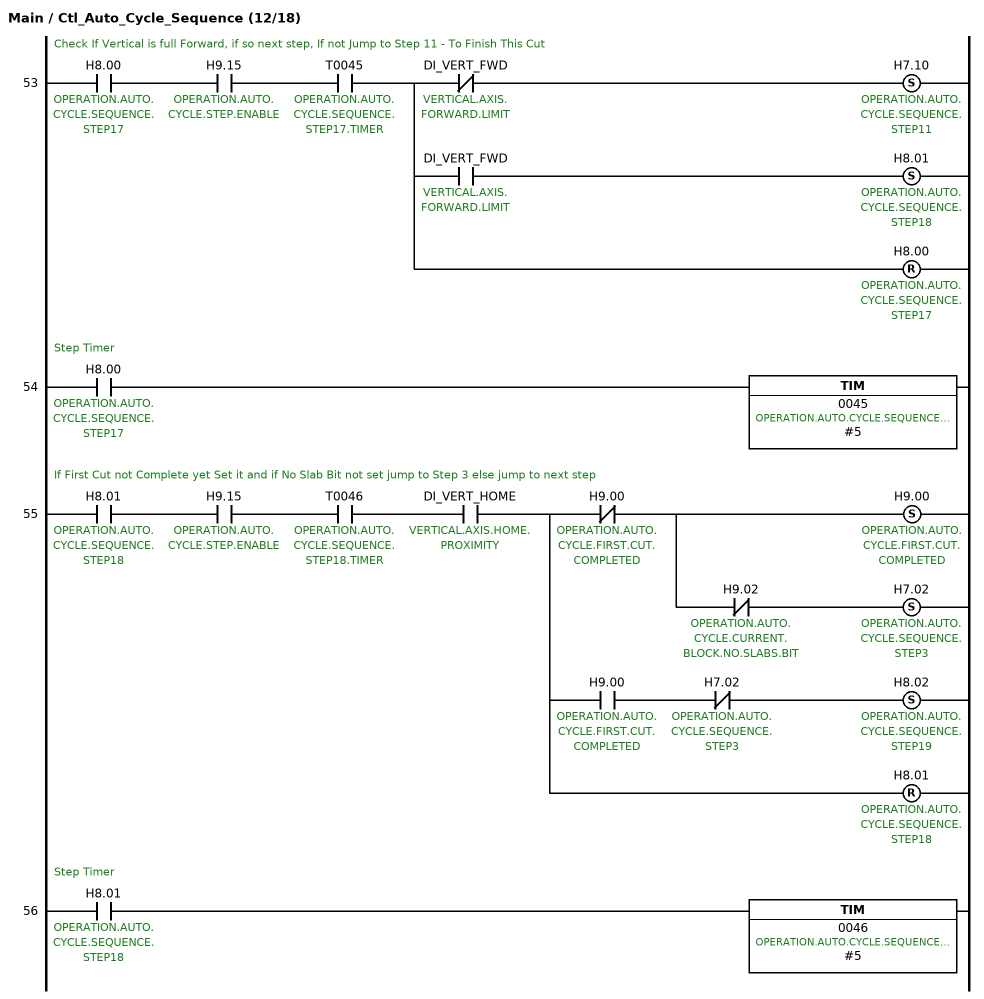
; [picture p24: Main / Ctl_Auto_Cycle_Sequence, rungs 53-56]
; rung 53: Check If Vertical is full Forward, if so next step, If not Jump to Step 11 - To Finish This Cut
LD H8.00  ; OPERATION.AUTO.CYCLE.SEQUENCE.STEP17
AND H9.15  ; OPERATION.AUTO.CYCLE.STEP.ENABLE
AND T0045  ; OPERATION.AUTO.CYCLE.SEQUENCE.STEP17.TIMER
OUT TR0
ANDNOT DI_VERT_FWD  ; VERTICAL.AXIS.FORWARD.LIMIT
SET H7.10  ; OPERATION.AUTO.CYCLE.SEQUENCE.STEP11
LD TR0
AND DI_VERT_FWD  ; VERTICAL.AXIS.FORWARD.LIMIT
SET H8.01  ; OPERATION.AUTO.CYCLE.SEQUENCE.STEP18
LD TR0
RSET H8.00  ; OPERATION.AUTO.CYCLE.SEQUENCE.STEP17
; rung 54: Step Timer
LD H8.00  ; OPERATION.AUTO.CYCLE.SEQUENCE.STEP17
TIM 0045 #5  ; OPERATION.AUTO.CYCLE.SEQUENCE.STEP17.TIMER
; rung 55: If First Cut not Complete yet Set it and if No Slab Bit not set jump to Step 3 else jump to next step
LD H8.01  ; OPERATION.AUTO.CYCLE.SEQUENCE.STEP18
AND H9.15  ; OPERATION.AUTO.CYCLE.STEP.ENABLE
AND T0046  ; OPERATION.AUTO.CYCLE.SEQUENCE.STEP18.TIMER
AND DI_VERT_HOME  ; VERTICAL.AXIS.HOME.PROXIMITY
OUT TR0
ANDNOT H9.00  ; OPERATION.AUTO.CYCLE.FIRST.CUT.COMPLETED
SET H9.00  ; OPERATION.AUTO.CYCLE.FIRST.CUT.COMPLETED
ANDNOT H9.02  ; OPERATION.AUTO.CYCLE.CURRENT.BLOCK.NO.SLABS.BIT
SET H7.02  ; OPERATION.AUTO.CYCLE.SEQUENCE.STEP3
LD TR0
AND H9.00  ; OPERATION.AUTO.CYCLE.FIRST.CUT.COMPLETED
ANDNOT H7.02  ; OPERATION.AUTO.CYCLE.SEQUENCE.STEP3
SET H8.02  ; OPERATION.AUTO.CYCLE.SEQUENCE.STEP19
LD TR0
RSET H8.01  ; OPERATION.AUTO.CYCLE.SEQUENCE.STEP18
; rung 56: Step Timer
LD H8.01  ; OPERATION.AUTO.CYCLE.SEQUENCE.STEP18
TIM 0046 #5  ; OPERATION.AUTO.CYCLE.SEQUENCE.STEP18.TIMER

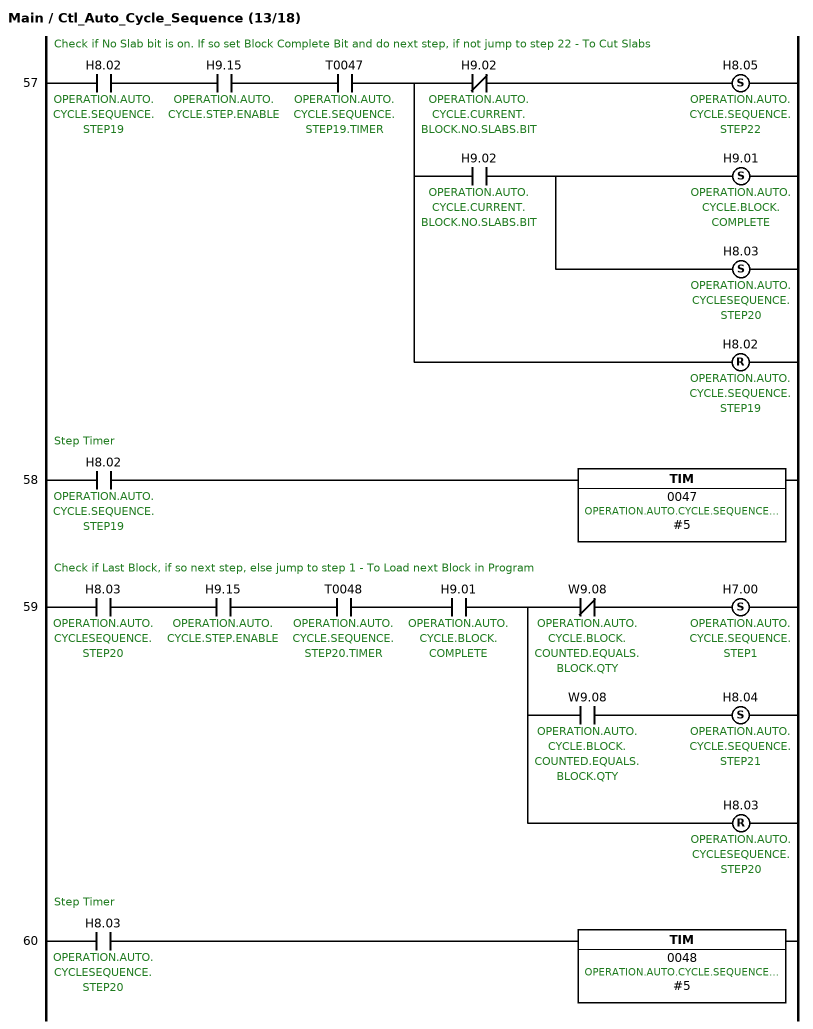
; rung 57: Check if No Slab bit is on. If so set Block Complete Bit and do next step, if not jump to step 22 - To Cut Slabs
LD H8.02  ; OPERATION.AUTO.CYCLE.SEQUENCE.STEP19
AND H9.15  ; OPERATION.AUTO.CYCLE.STEP.ENABLE
AND T0047  ; OPERATION.AUTO.CYCLE.SEQUENCE.STEP19.TIMER
OUT TR0
ANDNOT H9.02  ; OPERATION.AUTO.CYCLE.CURRENT.BLOCK.NO.SLABS.BIT
SET H8.05  ; OPERATION.AUTO.CYCLE.SEQUENCE.STEP22
LD TR0
AND H9.02  ; OPERATION.AUTO.CYCLE.CURRENT.BLOCK.NO.SLABS.BIT
SET H9.01  ; OPERATION.AUTO.CYCLE.BLOCK.COMPLETE
SET H8.03  ; OPERATION.AUTO.CYCLESEQUENCE.STEP20
LD TR0
RSET H8.02  ; OPERATION.AUTO.CYCLE.SEQUENCE.STEP19
; rung 58: Step Timer
LD H8.02  ; OPERATION.AUTO.CYCLE.SEQUENCE.STEP19
TIM 0047 #5  ; OPERATION.AUTO.CYCLE.SEQUENCE.STEP19.TIMER
; rung 59: Check if Last Block, if so next step, else jump to step 1 - To Load next Block in Program
LD H8.03  ; OPERATION.AUTO.CYCLESEQUENCE.STEP20
AND H9.15  ; OPERATION.AUTO.CYCLE.STEP.ENABLE
AND T0048  ; OPERATION.AUTO.CYCLE.SEQUENCE.STEP20.TIMER
AND H9.01  ; OPERATION.AUTO.CYCLE.BLOCK.COMPLETE
OUT TR0
ANDNOT W9.08  ; OPERATION.AUTO.CYCLE.BLOCK.COUNTED.EQUALS.BLOCK.QTY
SET H7.00  ; OPERATION.AUTO.CYCLE.SEQUENCE.STEP1
LD TR0
AND W9.08  ; OPERATION.AUTO.CYCLE.BLOCK.COUNTED.EQUALS.BLOCK.QTY
SET H8.04  ; OPERATION.AUTO.CYCLE.SEQUENCE.STEP21
LD TR0
RSET H8.03  ; OPERATION.AUTO.CYCLESEQUENCE.STEP20
; rung 60: Step Timer
LD H8.03  ; OPERATION.AUTO.CYCLESEQUENCE.STEP20
TIM 0048 #5  ; OPERATION.AUTO.CYCLE.SEQUENCE.STEP20.TIMER

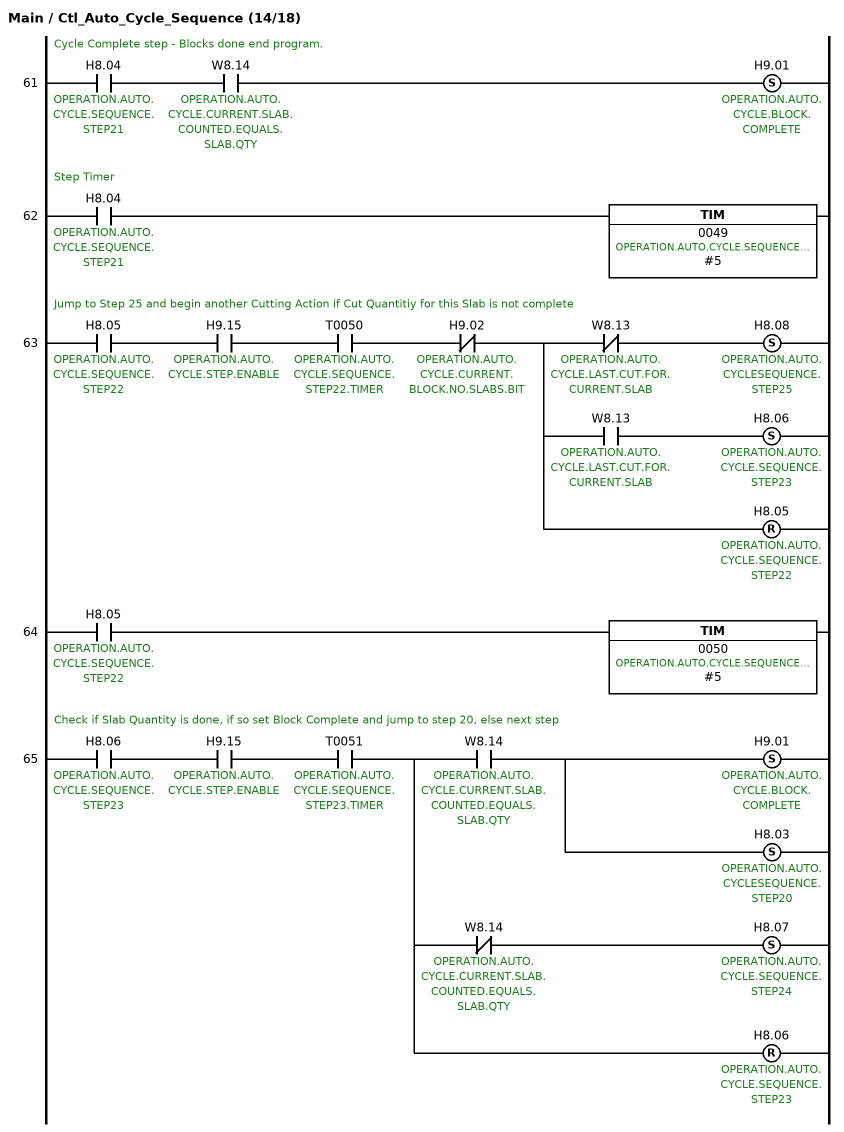
; rung 61: Cycle Complete step - Blocks done end program.
LD H8.04  ; OPERATION.AUTO.CYCLE.SEQUENCE.STEP21
AND W8.14  ; OPERATION.AUTO.CYCLE.CURRENT.SLAB.COUNTED.EQUALS.SLAB.QTY
SET H9.01  ; OPERATION.AUTO.CYCLE.BLOCK.COMPLETE
; rung 62: Step Timer
LD H8.04  ; OPERATION.AUTO.CYCLE.SEQUENCE.STEP21
TIM 0049 #5  ; OPERATION.AUTO.CYCLE.SEQUENCE.STEP21.TIMER
; rung 63: Jump to Step 25 and begin another Cutting Action if Cut Quantitiy for this Slab is not complete
LD H8.05  ; OPERATION.AUTO.CYCLE.SEQUENCE.STEP22
AND H9.15  ; OPERATION.AUTO.CYCLE.STEP.ENABLE
AND T0050  ; OPERATION.AUTO.CYCLE.SEQUENCE.STEP22.TIMER
ANDNOT H9.02  ; OPERATION.AUTO.CYCLE.CURRENT.BLOCK.NO.SLABS.BIT
OUT TR0
ANDNOT W8.13  ; OPERATION.AUTO.CYCLE.LAST.CUT.FOR.CURRENT.SLAB
SET H8.08  ; OPERATION.AUTO.CYCLESEQUENCE.STEP25
LD TR0
AND W8.13  ; OPERATION.AUTO.CYCLE.LAST.CUT.FOR.CURRENT.SLAB
SET H8.06  ; OPERATION.AUTO.CYCLE.SEQUENCE.STEP23
LD TR0
RSET H8.05  ; OPERATION.AUTO.CYCLE.SEQUENCE.STEP22
; rung 64
LD H8.05  ; OPERATION.AUTO.CYCLE.SEQUENCE.STEP22
TIM 0050 #5  ; OPERATION.AUTO.CYCLE.SEQUENCE.STEP22.TIMER
; rung 65: Check if Slab Quantity is done, if so set Block Complete and jump to step 20, else next step
LD H8.06  ; OPERATION.AUTO.CYCLE.SEQUENCE.STEP23
AND H9.15  ; OPERATION.AUTO.CYCLE.STEP.ENABLE
AND T0051  ; OPERATION.AUTO.CYCLE.SEQUENCE.STEP23.TIMER
OUT TR0
AND W8.14  ; OPERATION.AUTO.CYCLE.CURRENT.SLAB.COUNTED.EQUALS.SLAB.QTY
SET H9.01  ; OPERATION.AUTO.CYCLE.BLOCK.COMPLETE
SET H8.03  ; OPERATION.AUTO.CYCLESEQUENCE.STEP20
LD TR0
ANDNOT W8.14  ; OPERATION.AUTO.CYCLE.CURRENT.SLAB.COUNTED.EQUALS.SLAB.QTY
SET H8.07  ; OPERATION.AUTO.CYCLE.SEQUENCE.STEP24
LD TR0
RSET H8.06  ; OPERATION.AUTO.CYCLE.SEQUENCE.STEP23

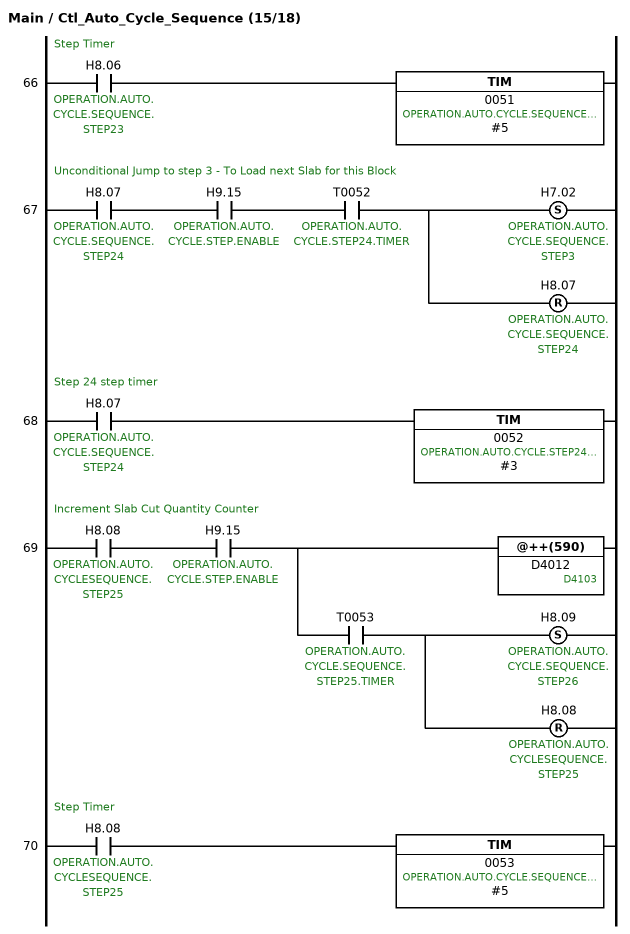
; rung 66: Step Timer
LD H8.06  ; OPERATION.AUTO.CYCLE.SEQUENCE.STEP23
TIM 0051 #5  ; OPERATION.AUTO.CYCLE.SEQUENCE.STEP23.TIMER
; rung 67: Unconditional Jump to step 3 - To Load next Slab for this Block
LD H8.07  ; OPERATION.AUTO.CYCLE.SEQUENCE.STEP24
AND H9.15  ; OPERATION.AUTO.CYCLE.STEP.ENABLE
AND T0052  ; OPERATION.AUTO.CYCLE.STEP24.TIMER
SET H7.02  ; OPERATION.AUTO.CYCLE.SEQUENCE.STEP3
RSET H8.07  ; OPERATION.AUTO.CYCLE.SEQUENCE.STEP24
; rung 68: Step 24 step timer
LD H8.07  ; OPERATION.AUTO.CYCLE.SEQUENCE.STEP24
TIM 0052 #3  ; OPERATION.AUTO.CYCLE.STEP24.TIMER
; rung 69: Increment Slab Cut Quantity Counter
LD H8.08  ; OPERATION.AUTO.CYCLESEQUENCE.STEP25
AND H9.15  ; OPERATION.AUTO.CYCLE.STEP.ENABLE
@++(590) D4012  ; D4103
AND T0053  ; OPERATION.AUTO.CYCLE.SEQUENCE.STEP25.TIMER
SET H8.09  ; OPERATION.AUTO.CYCLE.SEQUENCE.STEP26
RSET H8.08  ; OPERATION.AUTO.CYCLESEQUENCE.STEP25
; rung 70: Step Timer
LD H8.08  ; OPERATION.AUTO.CYCLESEQUENCE.STEP25
TIM 0053 #5  ; OPERATION.AUTO.CYCLE.SEQUENCE.STEP25.TIMER

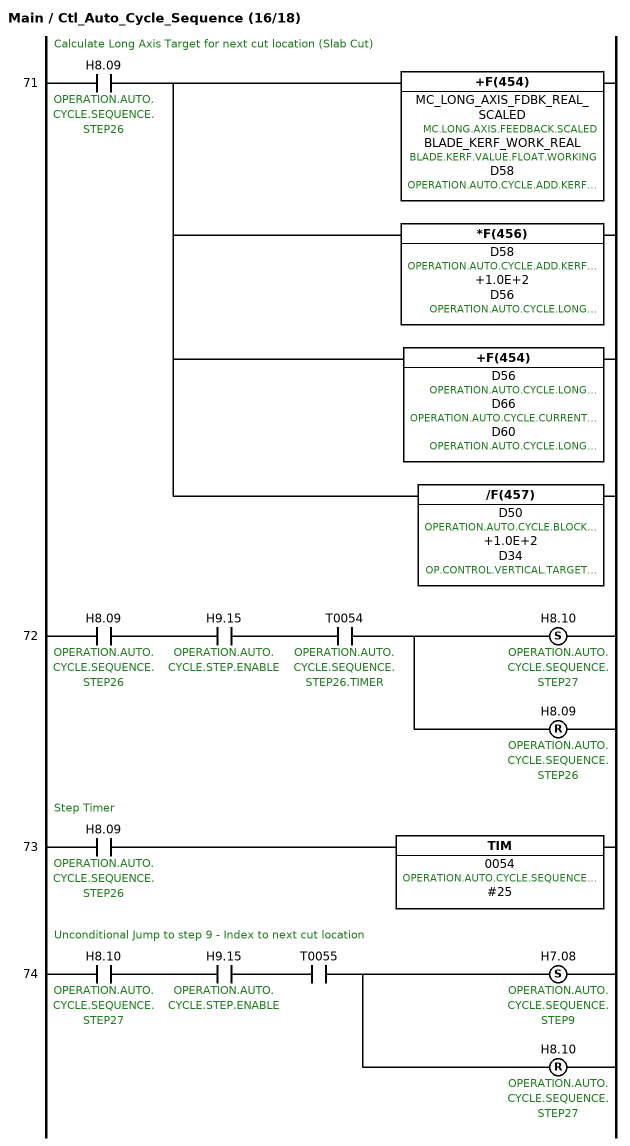
; rung 71: Calculate Long Axis Target for next cut location (Slab Cut)
LD H8.09  ; OPERATION.AUTO.CYCLE.SEQUENCE.STEP26
+F(454) MC_LONG_AXIS_FDBK_REAL_SCALED BLADE_KERF_WORK_REAL D58  ; MC.LONG.AXIS.FEEDBACK.SCALED, BLADE.KERF.VALUE.FLOAT.WORKING, OPERATION.AUTO.CYCLE.ADD.KERF.TO.LOCATION.REAL
*F(456) D58 +1.0E+2 D56  ; OPERATION.AUTO.CYCLE.ADD.KERF.TO.LOCATION.REAL, OPERATION.AUTO.CYCLE.LONG.TARGET.KERF
+F(454) D56 D66 D60  ; OPERATION.AUTO.CYCLE.LONG.TARGET.KERF, OPERATION.AUTO.CYCLE.CURRENT.SLAB.SIZE.REAL.RAW, OPERATION.AUTO.CYCLE.LONG.INDEX.LOCATION.REAL
/F(457) D50 +1.0E+2 D34  ; OPERATION.AUTO.CYCLE.BLOCK.HEIGHT.REAL, OP.CONTROL.VERTICAL.TARGET.SCALED
; rung 72
LD H8.09  ; OPERATION.AUTO.CYCLE.SEQUENCE.STEP26
AND H9.15  ; OPERATION.AUTO.CYCLE.STEP.ENABLE
AND T0054  ; OPERATION.AUTO.CYCLE.SEQUENCE.STEP26.TIMER
SET H8.10  ; OPERATION.AUTO.CYCLE.SEQUENCE.STEP27
RSET H8.09  ; OPERATION.AUTO.CYCLE.SEQUENCE.STEP26
; rung 73: Step Timer
LD H8.09  ; OPERATION.AUTO.CYCLE.SEQUENCE.STEP26
TIM 0054 #25  ; OPERATION.AUTO.CYCLE.SEQUENCE.STEP26.TIMER
; rung 74: Unconditional Jump to step 9 - Index to next cut location
LD H8.10  ; OPERATION.AUTO.CYCLE.SEQUENCE.STEP27
AND H9.15  ; OPERATION.AUTO.CYCLE.STEP.ENABLE
AND T0055
SET H7.08  ; OPERATION.AUTO.CYCLE.SEQUENCE.STEP9
RSET H8.10  ; OPERATION.AUTO.CYCLE.SEQUENCE.STEP27

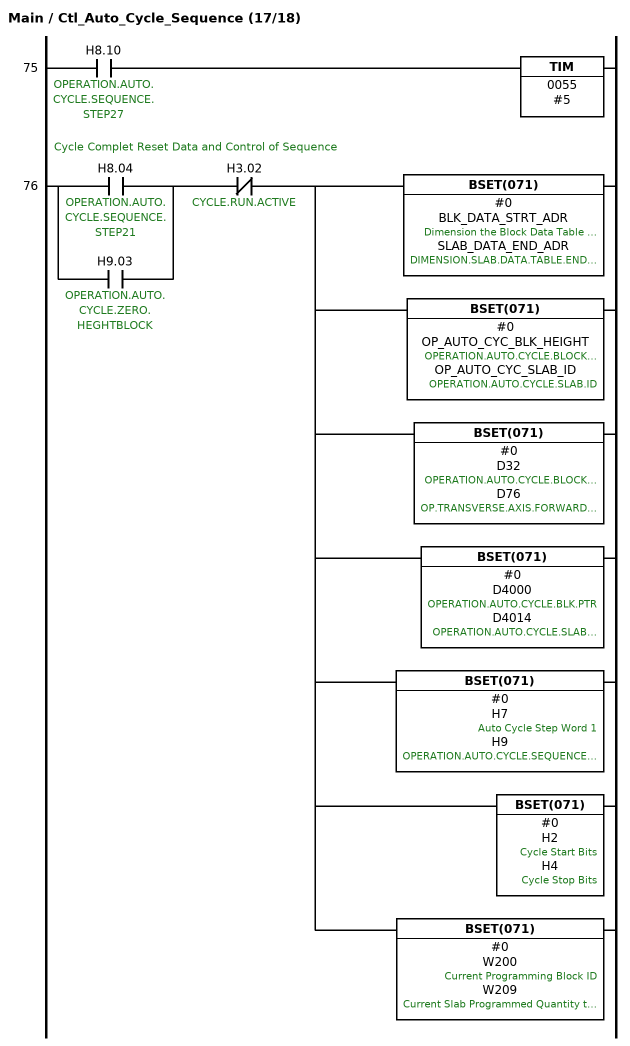
; rung 75
LD H8.10  ; OPERATION.AUTO.CYCLE.SEQUENCE.STEP27
TIM 0055 #5
; rung 76: Cycle Complet Reset Data and Control of Sequence
LD H8.04  ; OPERATION.AUTO.CYCLE.SEQUENCE.STEP21
OR H9.03  ; OPERATION.AUTO.CYCLE.ZERO.HEGHTBLOCK
ANDNOT H3.02  ; CYCLE.RUN.ACTIVE
BSET(071) #0 BLK_DATA_STRT_ADR SLAB_DATA_END_ADR  ; Dimension the Block Data Table - Start Address, DIMENSION.SLAB.DATA.TABLE.END.ADDRESS
BSET(071) #0 OP_AUTO_CYC_BLK_HEIGHT OP_AUTO_CYC_SLAB_ID  ; OPERATION.AUTO.CYCLE.BLOCK.HEIGHT.WORKING, OPERATION.AUTO.CYCLE.SLAB.ID
BSET(071) #0 D32 D76  ; OPERATION.AUTO.CYCLE.BLOCK.FIRST.CUT.WORKING.REAL, OP.TRANSVERSE.AXIS.FORWARD.TARGET
BSET(071) #0 D4000 D4014  ; OPERATION.AUTO.CYCLE.BLK.PTR, OPERATION.AUTO.CYCLE.SLAB.POINTER
BSET(071) #0 H7 H9  ; Auto Cycle Step Word 1, OPERATION.AUTO.CYCLE.SEQUENCE.STATE.BITS
BSET(071) #0 H2 H4  ; Cycle Start Bits, Cycle Stop Bits
BSET(071) #0 W200 W209  ; Current Programming Block ID, Current Slab Programmed Quantity to cut

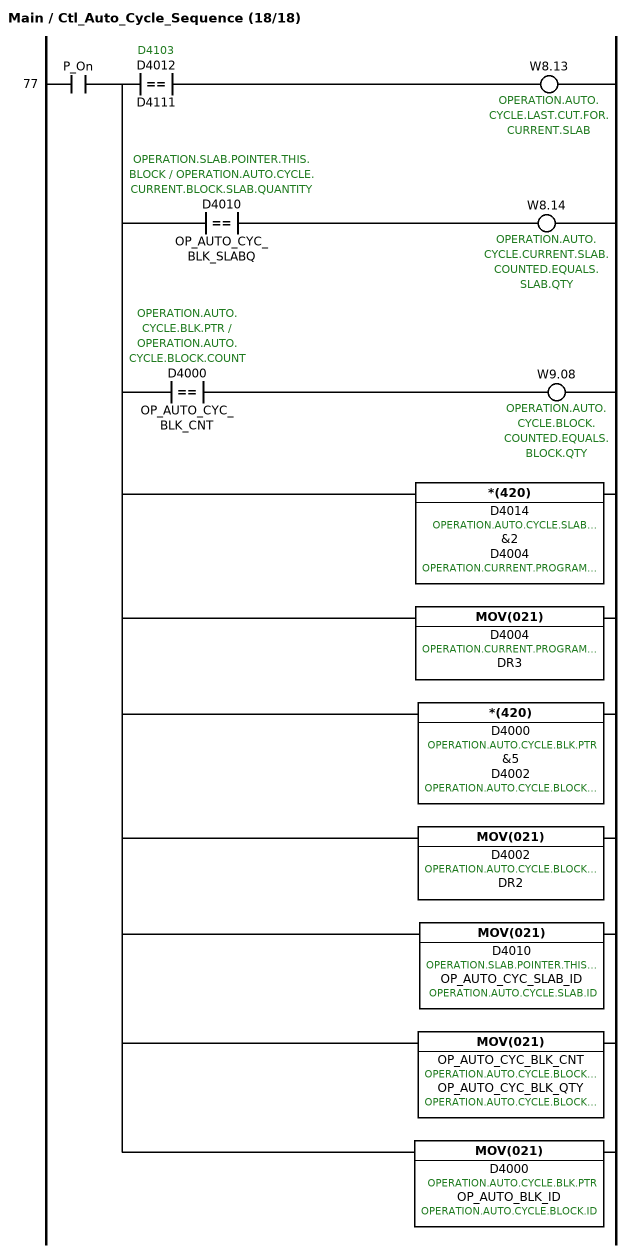
; rung 77
LD P_On
OUT TR0
AND=(300) D4012 D4111  ; D4103
OUT W8.13  ; OPERATION.AUTO.CYCLE.LAST.CUT.FOR.CURRENT.SLAB
LD TR0
AND=(300) D4010 OP_AUTO_CYC_BLK_SLABQ  ; OPERATION.SLAB.POINTER.THIS.BLOCK, OPERATION.AUTO.CYCLE.CURRENT.BLOCK.SLAB.QUANTITY
OUT W8.14  ; OPERATION.AUTO.CYCLE.CURRENT.SLAB.COUNTED.EQUALS.SLAB.QTY
LD TR0
AND=(300) D4000 OP_AUTO_CYC_BLK_CNT  ; OPERATION.AUTO.CYCLE.BLK.PTR, OPERATION.AUTO.CYCLE.BLOCK.COUNT
OUT W9.08  ; OPERATION.AUTO.CYCLE.BLOCK.COUNTED.EQUALS.BLOCK.QTY
LD TR0
*(420) D4014 &2 D4004  ; OPERATION.AUTO.CYCLE.SLAB.POINTER, OPERATION.CURRENT.PROGRAM.SLAB.DATA.POINTER
MOV(021) D4004 DR3  ; OPERATION.CURRENT.PROGRAM.SLAB.DATA.POINTER
*(420) D4000 &5 D4002  ; OPERATION.AUTO.CYCLE.BLK.PTR, OPERATION.AUTO.CYCLE.BLOCK.DATA.POINTER
MOV(021) D4002 DR2  ; OPERATION.AUTO.CYCLE.BLOCK.DATA.POINTER
MOV(021) D4010 OP_AUTO_CYC_SLAB_ID  ; OPERATION.SLAB.POINTER.THIS.BLOCK, OPERATION.AUTO.CYCLE.SLAB.ID
MOV(021) OP_AUTO_CYC_BLK_CNT OP_AUTO_CYC_BLK_QTY  ; OPERATION.AUTO.CYCLE.BLOCK.COUNT, OPERATION.AUTO.CYCLE.BLOCK.QUANTITY
MOV(021) D4000 OP_AUTO_BLK_ID  ; OPERATION.AUTO.CYCLE.BLK.PTR, OPERATION.AUTO.CYCLE.BLOCK.ID

### Section Ctl_Master_Home

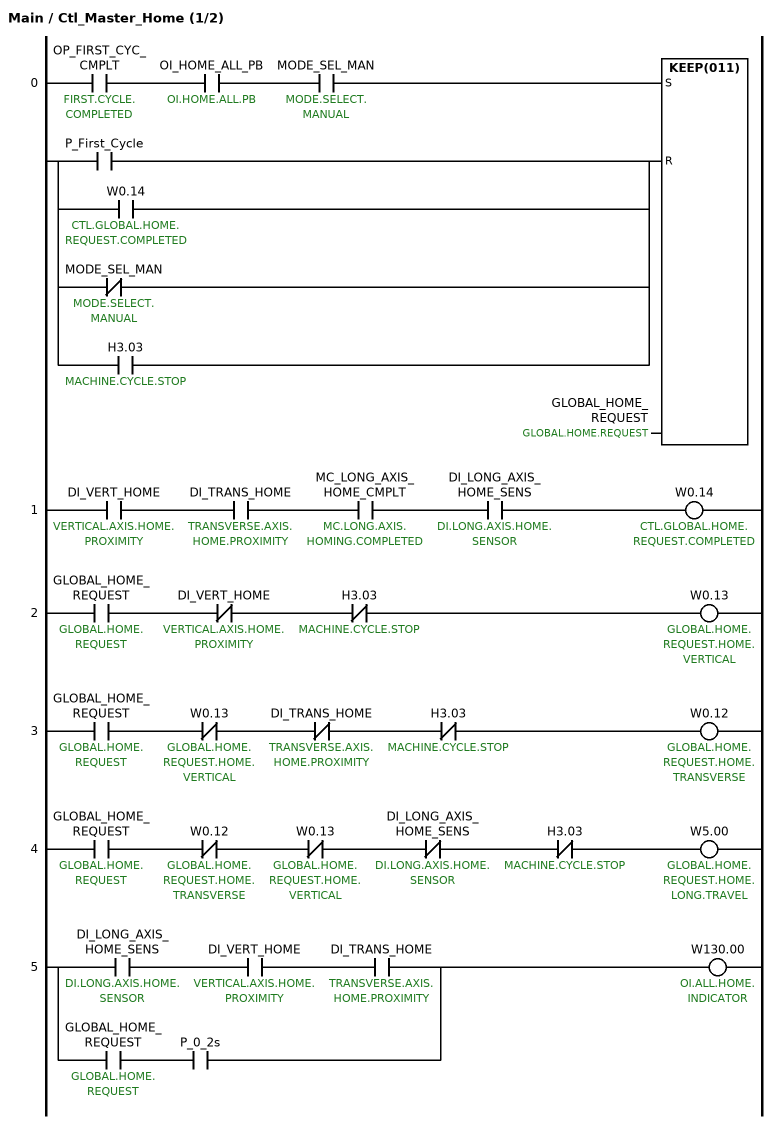
; rung 0
LD OP_FIRST_CYC_CMPLT  ; FIRST.CYCLE.COMPLETED
AND OI_HOME_ALL_PB  ; OI.HOME.ALL.PB
AND MODE_SEL_MAN  ; MODE.SELECT.MANUAL
LD P_First_Cycle
OR W0.14  ; CTL.GLOBAL.HOME.REQUEST.COMPLETED
ORNOT MODE_SEL_MAN  ; MODE.SELECT.MANUAL
OR H3.03  ; MACHINE.CYCLE.STOP
KEEP(011) GLOBAL_HOME_REQUEST  ; GLOBAL.HOME.REQUEST
; rung 1
LD DI_VERT_HOME  ; VERTICAL.AXIS.HOME.PROXIMITY
AND DI_TRANS_HOME  ; TRANSVERSE.AXIS.HOME.PROXIMITY
AND MC_LONG_AXIS_HOME_CMPLT  ; MC.LONG.AXIS.HOMING.COMPLETED
AND DI_LONG_AXIS_HOME_SENS  ; DI.LONG.AXIS.HOME.SENSOR
OUT W0.14  ; CTL.GLOBAL.HOME.REQUEST.COMPLETED
; rung 2
LD GLOBAL_HOME_REQUEST  ; GLOBAL.HOME.REQUEST
ANDNOT DI_VERT_HOME  ; VERTICAL.AXIS.HOME.PROXIMITY
ANDNOT H3.03  ; MACHINE.CYCLE.STOP
OUT W0.13  ; GLOBAL.HOME.REQUEST.HOME.VERTICAL
; rung 3
LD GLOBAL_HOME_REQUEST  ; GLOBAL.HOME.REQUEST
ANDNOT W0.13  ; GLOBAL.HOME.REQUEST.HOME.VERTICAL
ANDNOT DI_TRANS_HOME  ; TRANSVERSE.AXIS.HOME.PROXIMITY
ANDNOT H3.03  ; MACHINE.CYCLE.STOP
OUT W0.12  ; GLOBAL.HOME.REQUEST.HOME.TRANSVERSE
; rung 4
LD GLOBAL_HOME_REQUEST  ; GLOBAL.HOME.REQUEST
ANDNOT W0.12  ; GLOBAL.HOME.REQUEST.HOME.TRANSVERSE
ANDNOT W0.13  ; GLOBAL.HOME.REQUEST.HOME.VERTICAL
ANDNOT DI_LONG_AXIS_HOME_SENS  ; DI.LONG.AXIS.HOME.SENSOR
ANDNOT H3.03  ; MACHINE.CYCLE.STOP
OUT W5.00  ; GLOBAL.HOME.REQUEST.HOME.LONG.TRAVEL
; rung 5
LD DI_LONG_AXIS_HOME_SENS  ; DI.LONG.AXIS.HOME.SENSOR
AND DI_VERT_HOME  ; VERTICAL.AXIS.HOME.PROXIMITY
AND DI_TRANS_HOME  ; TRANSVERSE.AXIS.HOME.PROXIMITY
LD GLOBAL_HOME_REQUEST  ; GLOBAL.HOME.REQUEST
AND P_0_2s
ORLD
OUT W130.00  ; OI.ALL.HOME.INDICATOR

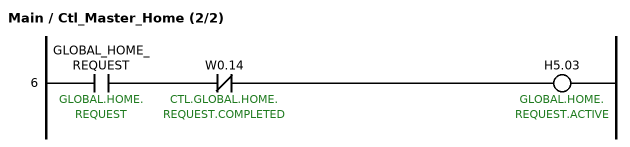
; rung 6
LD GLOBAL_HOME_REQUEST  ; GLOBAL.HOME.REQUEST
ANDNOT W0.14  ; CTL.GLOBAL.HOME.REQUEST.COMPLETED
OUT H5.03  ; GLOBAL.HOME.REQUEST.ACTIVE

### Section Ctl_Long_Axis

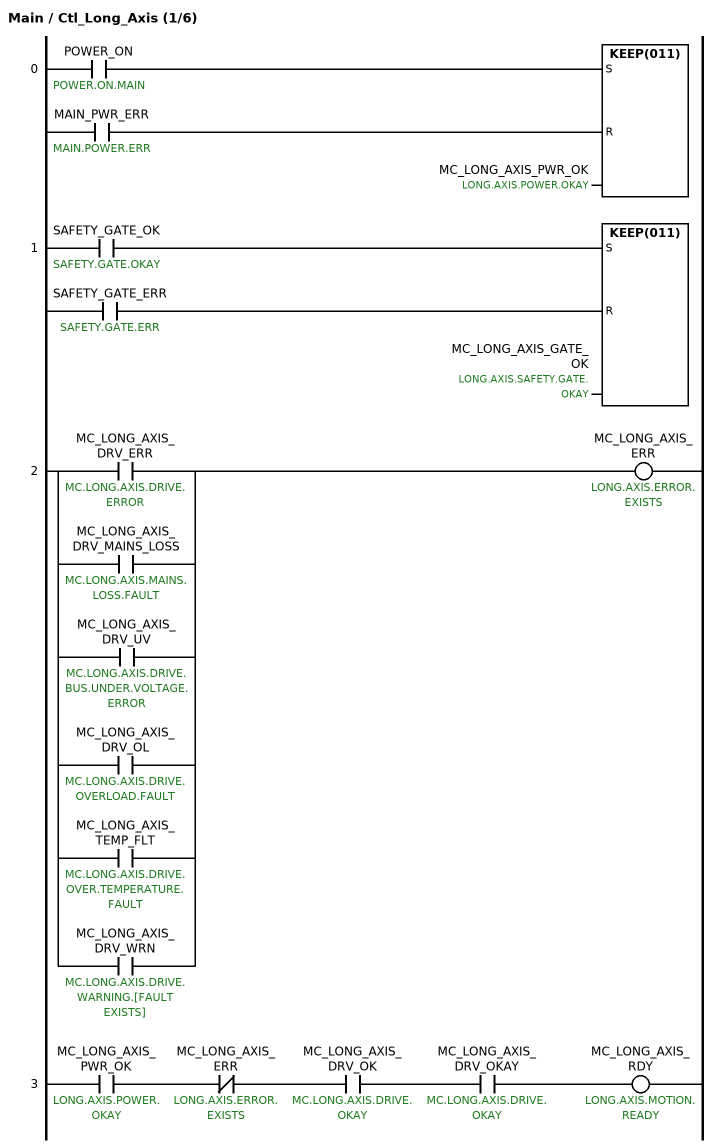
; rung 0
LD POWER_ON  ; POWER.ON.MAIN
LD MAIN_PWR_ERR  ; MAIN.POWER.ERR
KEEP(011) MC_LONG_AXIS_PWR_OK  ; LONG.AXIS.POWER.OKAY
; rung 1
LD SAFETY_GATE_OK  ; SAFETY.GATE.OKAY
LD SAFETY_GATE_ERR  ; SAFETY.GATE.ERR
KEEP(011) MC_LONG_AXIS_GATE_OK  ; LONG.AXIS.SAFETY.GATE.OKAY
; rung 2
LD MC_LONG_AXIS_DRV_ERR  ; MC.LONG.AXIS.DRIVE.ERROR
OR MC_LONG_AXIS_DRV_MAINS_LOSS  ; MC.LONG.AXIS.MAINS.LOSS.FAULT
OR MC_LONG_AXIS_DRV_UV  ; MC.LONG.AXIS.DRIVE.BUS.UNDER.VOLTAGE.ERROR
OR MC_LONG_AXIS_DRV_OL  ; MC.LONG.AXIS.DRIVE.OVERLOAD.FAULT
OR MC_LONG_AXIS_TEMP_FLT  ; MC.LONG.AXIS.DRIVE.OVER.TEMPERATURE.FAULT
OR MC_LONG_AXIS_DRV_WRN  ; MC.LONG.AXIS.DRIVE.WARNING.[FAULT EXISTS]
OUT MC_LONG_AXIS_ERR  ; LONG.AXIS.ERROR.EXISTS
; rung 3
LD MC_LONG_AXIS_PWR_OK  ; LONG.AXIS.POWER.OKAY
ANDNOT MC_LONG_AXIS_ERR  ; LONG.AXIS.ERROR.EXISTS
AND MC_LONG_AXIS_DRV_OK  ; MC.LONG.AXIS.DRIVE.OKAY
AND MC_LONG_AXIS_DRV_OKAY  ; MC.LONG.AXIS.DRIVE.OKAY
OUT MC_LONG_AXIS_RDY  ; LONG.AXIS.MOTION.READY

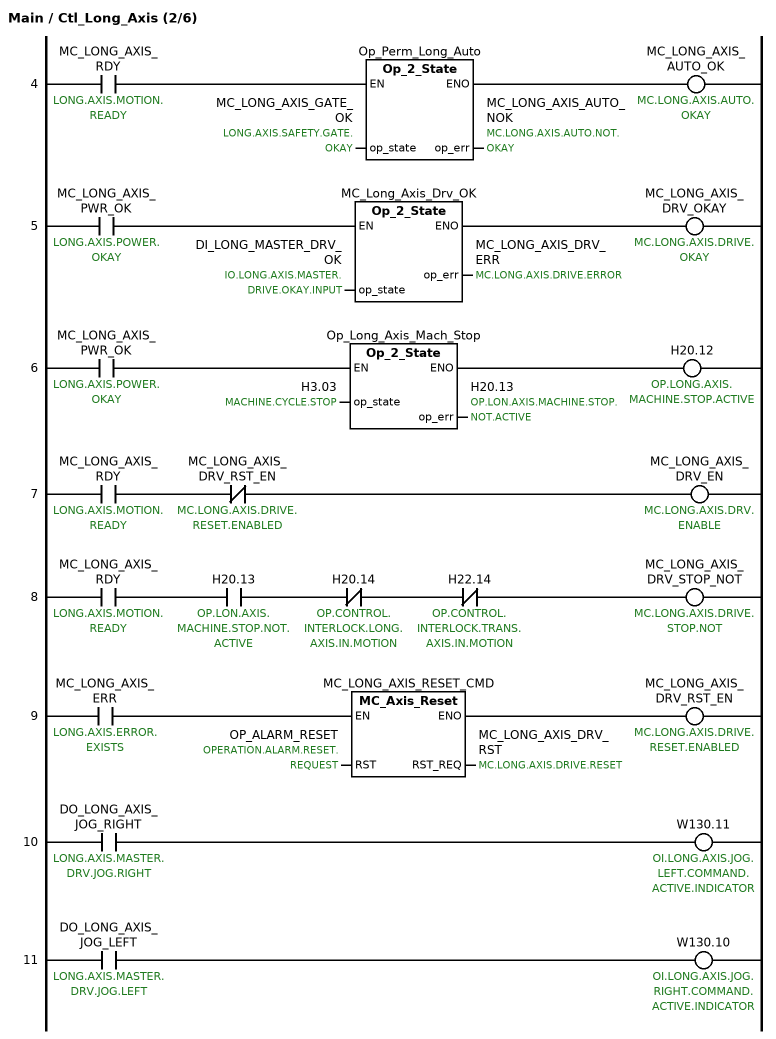
; rung 4
LD MC_LONG_AXIS_RDY  ; LONG.AXIS.MOTION.READY
CALL Op_Perm_Long_Auto : Op_2_State (op_state := MC_LONG_AXIS_GATE_OK, op_err => MC_LONG_AXIS_AUTO_NOK)  ; LONG.AXIS.SAFETY.GATE.OKAY, MC.LONG.AXIS.AUTO.NOT.OKAY
OUT MC_LONG_AXIS_AUTO_OK  ; MC.LONG.AXIS.AUTO.OKAY
; rung 5
LD MC_LONG_AXIS_PWR_OK  ; LONG.AXIS.POWER.OKAY
CALL MC_Long_Axis_Drv_OK : Op_2_State (op_state := DI_LONG_MASTER_DRV_OK, op_err => MC_LONG_AXIS_DRV_ERR)  ; IO.LONG.AXIS.MASTER.DRIVE.OKAY.INPUT, MC.LONG.AXIS.DRIVE.ERROR
OUT MC_LONG_AXIS_DRV_OKAY  ; MC.LONG.AXIS.DRIVE.OKAY
; rung 6
LD MC_LONG_AXIS_PWR_OK  ; LONG.AXIS.POWER.OKAY
CALL Op_Long_Axis_Mach_Stop : Op_2_State (op_state := H3.03, op_err => H20.13)  ; MACHINE.CYCLE.STOP, OP.LON.AXIS.MACHINE.STOP.NOT.ACTIVE
OUT H20.12  ; OP.LONG.AXIS.MACHINE.STOP.ACTIVE
; rung 7
LD MC_LONG_AXIS_RDY  ; LONG.AXIS.MOTION.READY
ANDNOT MC_LONG_AXIS_DRV_RST_EN  ; MC.LONG.AXIS.DRIVE.RESET.ENABLED
OUT MC_LONG_AXIS_DRV_EN  ; MC.LONG.AXIS.DRV.ENABLE
; rung 8
LD MC_LONG_AXIS_RDY  ; LONG.AXIS.MOTION.READY
AND H20.13  ; OP.LON.AXIS.MACHINE.STOP.NOT.ACTIVE
ANDNOT H20.14  ; OP.CONTROL.INTERLOCK.LONG.AXIS.IN.MOTION
ANDNOT H22.14  ; OP.CONTROL.INTERLOCK.TRANS.AXIS.IN.MOTION
OUT MC_LONG_AXIS_DRV_STOP_NOT  ; MC.LONG.AXIS.DRIVE.STOP.NOT
; rung 9
LD MC_LONG_AXIS_ERR  ; LONG.AXIS.ERROR.EXISTS
CALL MC_LONG_AXIS_RESET_CMD : MC_Axis_Reset (RST := OP_ALARM_RESET, RST_REQ => MC_LONG_AXIS_DRV_RST)  ; OPERATION.ALARM.RESET.REQUEST, MC.LONG.AXIS.DRIVE.RESET
OUT MC_LONG_AXIS_DRV_RST_EN  ; MC.LONG.AXIS.DRIVE.RESET.ENABLED
; rung 10
LD DO_LONG_AXIS_JOG_RIGHT  ; LONG.AXIS.MASTER.DRV.JOG.RIGHT
OUT W130.11  ; OI.LONG.AXIS.JOG.LEFT.COMMAND.ACTIVE.INDICATOR
; rung 11
LD DO_LONG_AXIS_JOG_LEFT  ; LONG.AXIS.MASTER.DRV.JOG.LEFT
OUT W130.10  ; OI.LONG.AXIS.JOG.RIGHT.COMMAND.ACTIVE.INDICATOR

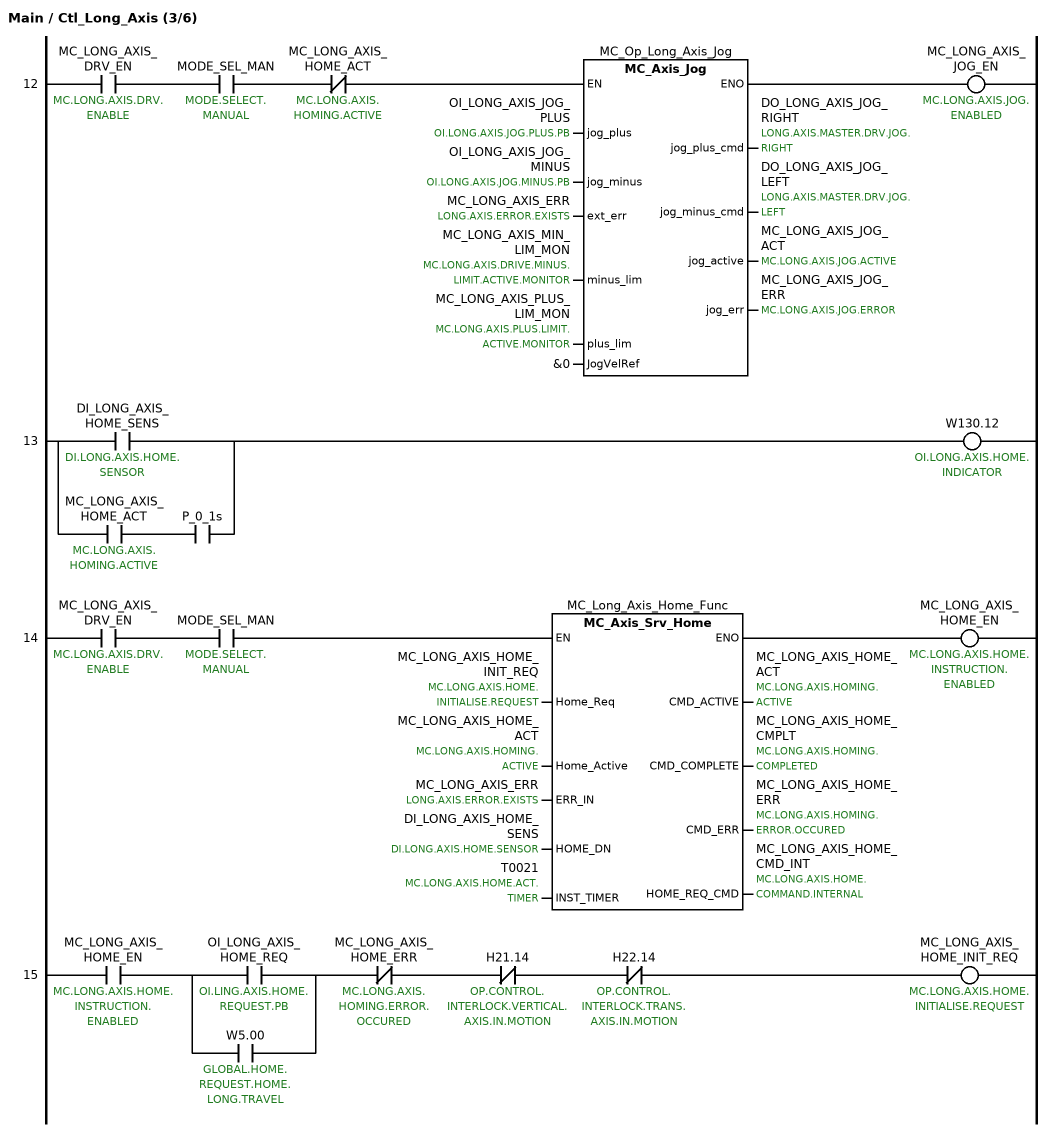
; rung 12
LD MC_LONG_AXIS_DRV_EN  ; MC.LONG.AXIS.DRV.ENABLE
AND MODE_SEL_MAN  ; MODE.SELECT.MANUAL
ANDNOT MC_LONG_AXIS_HOME_ACT  ; MC.LONG.AXIS.HOMING.ACTIVE
CALL MC_Op_Long_Axis_Jog : MC_Axis_Jog (jog_plus := OI_LONG_AXIS_JOG_PLUS, jog_minus := OI_LONG_AXIS_JOG_MINUS, ext_err := MC_LONG_AXIS_ERR, minus_lim := MC_LONG_AXIS_MIN_LIM_MON, plus_lim := MC_LONG_AXIS_PLUS_LIM_MON, JogVelRef := &0, jog_plus_cmd => DO_LONG_AXIS_JOG_RIGHT, jog_minus_cmd => DO_LONG_AXIS_JOG_LEFT, jog_active => MC_LONG_AXIS_JOG_ACT, jog_err => MC_LONG_AXIS_JOG_ERR)  ; OI.LONG.AXIS.JOG.PLUS.PB, OI.LONG.AXIS.JOG.MINUS.PB, LONG.AXIS.ERROR.EXISTS, MC.LONG.AXIS.DRIVE.MINUS.LIMIT.ACTIVE.MONITOR, MC.LONG.AXIS.PLUS.LIMIT.ACTIVE.MONITOR, LONG.AXIS.MASTER.DRV.JOG.RIGHT, LONG.AXIS.MASTER.DRV.JOG.LEFT, MC.LONG.AXIS.JOG.ACTIVE, MC.LONG.AXIS.JOG.ERROR
OUT MC_LONG_AXIS_JOG_EN  ; MC.LONG.AXIS.JOG.ENABLED
; rung 13
LD DI_LONG_AXIS_HOME_SENS  ; DI.LONG.AXIS.HOME.SENSOR
LD MC_LONG_AXIS_HOME_ACT  ; MC.LONG.AXIS.HOMING.ACTIVE
AND P_0_1s
ORLD
OUT W130.12  ; OI.LONG.AXIS.HOME.INDICATOR
; rung 14
LD MC_LONG_AXIS_DRV_EN  ; MC.LONG.AXIS.DRV.ENABLE
AND MODE_SEL_MAN  ; MODE.SELECT.MANUAL
CALL MC_Long_Axis_Home_Func : MC_Axis_Srv_Home (Home_Req := MC_LONG_AXIS_HOME_INIT_REQ, Home_Active := MC_LONG_AXIS_HOME_ACT, ERR_IN := MC_LONG_AXIS_ERR, HOME_DN := DI_LONG_AXIS_HOME_SENS, INST_TIMER := T0021, CMD_ACTIVE => MC_LONG_AXIS_HOME_ACT, CMD_COMPLETE => MC_LONG_AXIS_HOME_CMPLT, CMD_ERR => MC_LONG_AXIS_HOME_ERR, HOME_REQ_CMD => MC_LONG_AXIS_HOME_CMD_INT)  ; MC.LONG.AXIS.HOME.INITIALISE.REQUEST, MC.LONG.AXIS.HOMING.ACTIVE, LONG.AXIS.ERROR.EXISTS, DI.LONG.AXIS.HOME.SENSOR, MC.LONG.AXIS.HOME.ACT.TIMER, MC.LONG.AXIS.HOMING.COMPLETED, MC.LONG.AXIS.HOMING.ERROR.OCCURED, MC.LONG.AXIS.HOME.COMMAND.INTERNAL
OUT MC_LONG_AXIS_HOME_EN  ; MC.LONG.AXIS.HOME.INSTRUCTION.ENABLED
; rung 15
LD MC_LONG_AXIS_HOME_EN  ; MC.LONG.AXIS.HOME.INSTRUCTION.ENABLED
LD OI_LONG_AXIS_HOME_REQ  ; OI.LING.AXIS.HOME.REQUEST.PB
OR W5.00  ; GLOBAL.HOME.REQUEST.HOME.LONG.TRAVEL
ANDLD
ANDNOT MC_LONG_AXIS_HOME_ERR  ; MC.LONG.AXIS.HOMING.ERROR.OCCURED
ANDNOT H21.14  ; OP.CONTROL.INTERLOCK.VERTICAL.AXIS.IN.MOTION
ANDNOT H22.14  ; OP.CONTROL.INTERLOCK.TRANS.AXIS.IN.MOTION
OUT MC_LONG_AXIS_HOME_INIT_REQ  ; MC.LONG.AXIS.HOME.INITIALISE.REQUEST

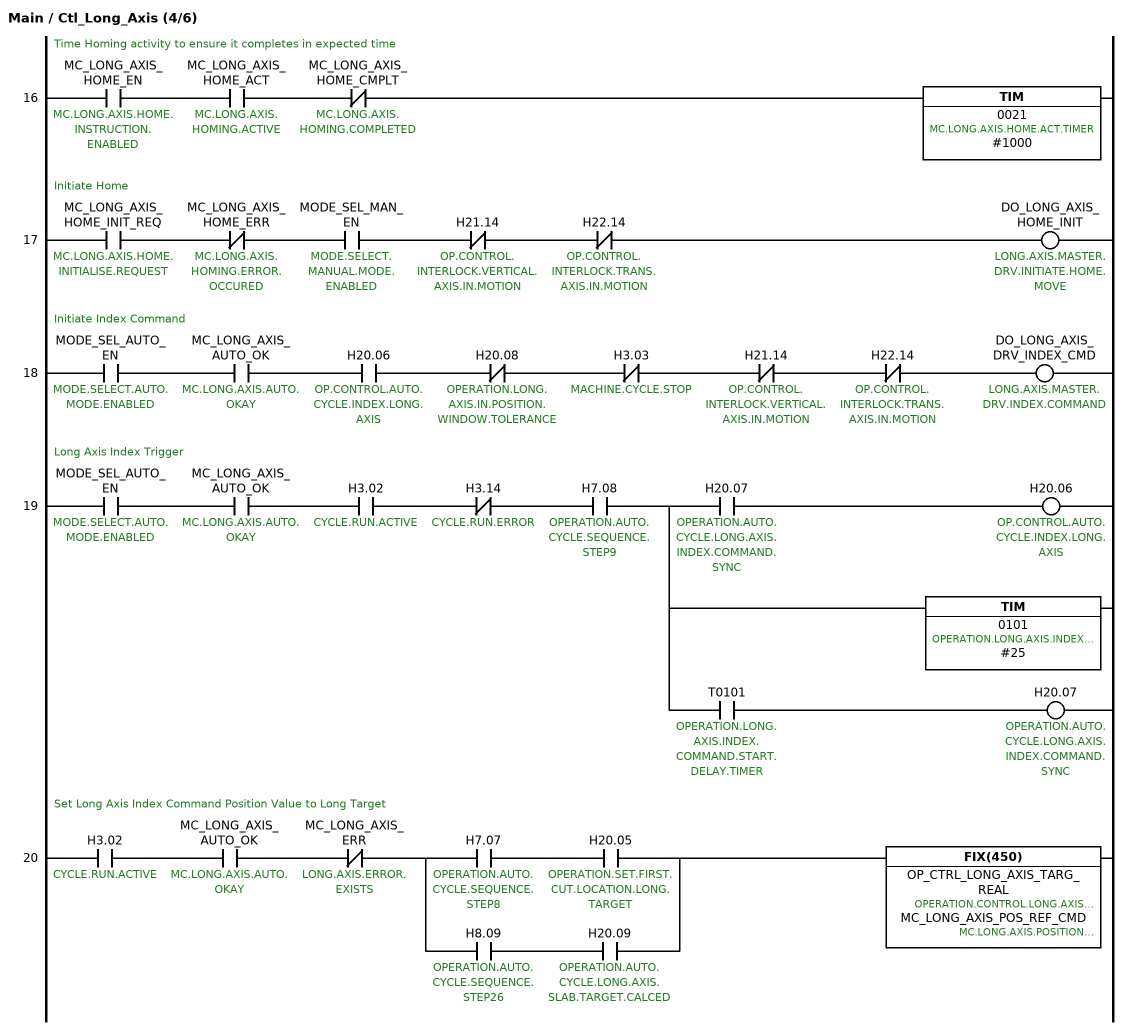
; rung 16: Time Homing activity to ensure it completes in expected time
LD MC_LONG_AXIS_HOME_EN  ; MC.LONG.AXIS.HOME.INSTRUCTION.ENABLED
AND MC_LONG_AXIS_HOME_ACT  ; MC.LONG.AXIS.HOMING.ACTIVE
ANDNOT MC_LONG_AXIS_HOME_CMPLT  ; MC.LONG.AXIS.HOMING.COMPLETED
TIM 0021 #1000  ; MC.LONG.AXIS.HOME.ACT.TIMER
; rung 17: Initiate Home
LD MC_LONG_AXIS_HOME_INIT_REQ  ; MC.LONG.AXIS.HOME.INITIALISE.REQUEST
ANDNOT MC_LONG_AXIS_HOME_ERR  ; MC.LONG.AXIS.HOMING.ERROR.OCCURED
AND MODE_SEL_MAN_EN  ; MODE.SELECT.MANUAL.MODE.ENABLED
ANDNOT H21.14  ; OP.CONTROL.INTERLOCK.VERTICAL.AXIS.IN.MOTION
ANDNOT H22.14  ; OP.CONTROL.INTERLOCK.TRANS.AXIS.IN.MOTION
OUT DO_LONG_AXIS_HOME_INIT  ; LONG.AXIS.MASTER.DRV.INITIATE.HOME.MOVE
; rung 18: Initiate Index Command
LD MODE_SEL_AUTO_EN  ; MODE.SELECT.AUTO.MODE.ENABLED
AND MC_LONG_AXIS_AUTO_OK  ; MC.LONG.AXIS.AUTO.OKAY
AND H20.06  ; OP.CONTROL.AUTO.CYCLE.INDEX.LONG.AXIS
ANDNOT H20.08  ; OPERATION.LONG.AXIS.IN.POSITION.WINDOW.TOLERANCE
ANDNOT H3.03  ; MACHINE.CYCLE.STOP
ANDNOT H21.14  ; OP.CONTROL.INTERLOCK.VERTICAL.AXIS.IN.MOTION
ANDNOT H22.14  ; OP.CONTROL.INTERLOCK.TRANS.AXIS.IN.MOTION
OUT DO_LONG_AXIS_DRV_INDEX_CMD  ; LONG.AXIS.MASTER.DRV.INDEX.COMMAND
; rung 19: Long Axis Index Trigger
LD MODE_SEL_AUTO_EN  ; MODE.SELECT.AUTO.MODE.ENABLED
AND MC_LONG_AXIS_AUTO_OK  ; MC.LONG.AXIS.AUTO.OKAY
AND H3.02  ; CYCLE.RUN.ACTIVE
ANDNOT H3.14  ; CYCLE.RUN.ERROR
AND H7.08  ; OPERATION.AUTO.CYCLE.SEQUENCE.STEP9
OUT TR0
AND H20.07  ; OPERATION.AUTO.CYCLE.LONG.AXIS.INDEX.COMMAND.SYNC
OUT H20.06  ; OP.CONTROL.AUTO.CYCLE.INDEX.LONG.AXIS
LD TR0
TIM 0101 #25  ; OPERATION.LONG.AXIS.INDEX.COMMAND.START.DELAY.TIMER
AND T0101  ; OPERATION.LONG.AXIS.INDEX.COMMAND.START.DELAY.TIMER
OUT H20.07  ; OPERATION.AUTO.CYCLE.LONG.AXIS.INDEX.COMMAND.SYNC
; rung 20: Set Long Axis Index Command Position Value to Long Target
LD H3.02  ; CYCLE.RUN.ACTIVE
AND MC_LONG_AXIS_AUTO_OK  ; MC.LONG.AXIS.AUTO.OKAY
ANDNOT MC_LONG_AXIS_ERR  ; LONG.AXIS.ERROR.EXISTS
LD H7.07  ; OPERATION.AUTO.CYCLE.SEQUENCE.STEP8
AND H20.05  ; OPERATION.SET.FIRST.CUT.LOCATION.LONG.TARGET
LD H8.09  ; OPERATION.AUTO.CYCLE.SEQUENCE.STEP26
AND H20.09  ; OPERATION.AUTO.CYCLE.LONG.AXIS.SLAB.TARGET.CALCED
ORLD
ANDLD
FIX(450) OP_CTRL_LONG_AXIS_TARG_REAL MC_LONG_AXIS_POS_REF_CMD  ; OPERATION.CONTROL.LONG.AXIS.TARGET.REAL, MC.LONG.AXIS.POSITION.REFERENCE.COMMAND.VALUE

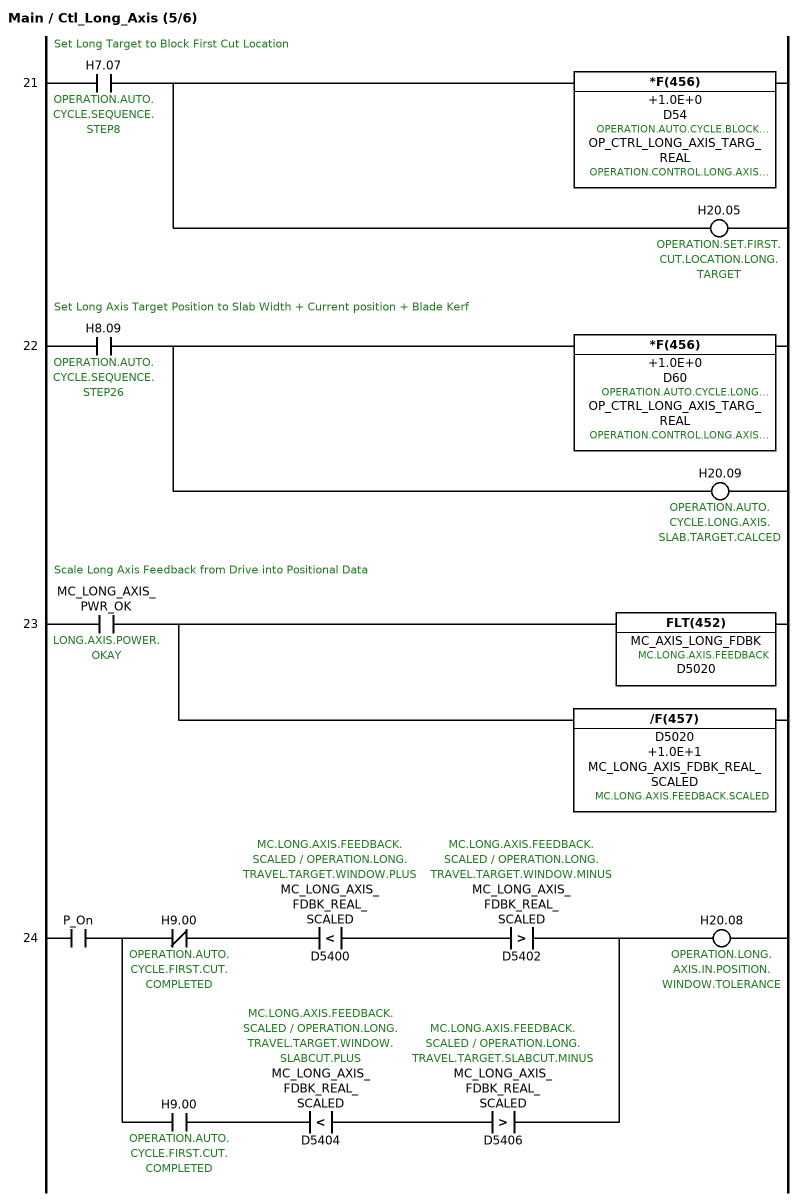
; rung 21: Set Long Target to Block First Cut Location
LD H7.07  ; OPERATION.AUTO.CYCLE.SEQUENCE.STEP8
*F(456) +1.0E+0 D54 OP_CTRL_LONG_AXIS_TARG_REAL  ; OPERATION.AUTO.CYCLE.BLOCK.FIRST.CUT.REAL, OPERATION.CONTROL.LONG.AXIS.TARGET.REAL
OUT H20.05  ; OPERATION.SET.FIRST.CUT.LOCATION.LONG.TARGET
; rung 22: Set Long Axis Target Position to Slab Width + Current position + Blade Kerf
LD H8.09  ; OPERATION.AUTO.CYCLE.SEQUENCE.STEP26
*F(456) +1.0E+0 D60 OP_CTRL_LONG_AXIS_TARG_REAL  ; OPERATION.AUTO.CYCLE.LONG.INDEX.LOCATION.REAL, OPERATION.CONTROL.LONG.AXIS.TARGET.REAL
OUT H20.09  ; OPERATION.AUTO.CYCLE.LONG.AXIS.SLAB.TARGET.CALCED
; rung 23: Scale Long Axis Feedback from Drive into Positional Data
LD MC_LONG_AXIS_PWR_OK  ; LONG.AXIS.POWER.OKAY
FLT(452) MC_AXIS_LONG_FDBK D5020  ; MC.LONG.AXIS.FEEDBACK
/F(457) D5020 +1.0E+1 MC_LONG_AXIS_FDBK_REAL_SCALED  ; MC.LONG.AXIS.FEEDBACK.SCALED
; rung 24
LD P_On
LDNOT H9.00  ; OPERATION.AUTO.CYCLE.FIRST.CUT.COMPLETED
AND<F(331) MC_LONG_AXIS_FDBK_REAL_SCALED D5400  ; MC.LONG.AXIS.FEEDBACK.SCALED, OPERATION.LONG.TRAVEL.TARGET.WINDOW.PLUS
AND>F(333) MC_LONG_AXIS_FDBK_REAL_SCALED D5402  ; MC.LONG.AXIS.FEEDBACK.SCALED, OPERATION.LONG.TRAVEL.TARGET.WINDOW.MINUS
LD H9.00  ; OPERATION.AUTO.CYCLE.FIRST.CUT.COMPLETED
AND<F(331) MC_LONG_AXIS_FDBK_REAL_SCALED D5404  ; MC.LONG.AXIS.FEEDBACK.SCALED, OPERATION.LONG.TRAVEL.TARGET.WINDOW.SLABCUT.PLUS
AND>F(333) MC_LONG_AXIS_FDBK_REAL_SCALED D5406  ; MC.LONG.AXIS.FEEDBACK.SCALED, OPERATION.LONG.TRAVEL.TARGET.SLABCUT.MINUS
ORLD
ANDLD
OUT H20.08  ; OPERATION.LONG.AXIS.IN.POSITION.WINDOW.TOLERANCE

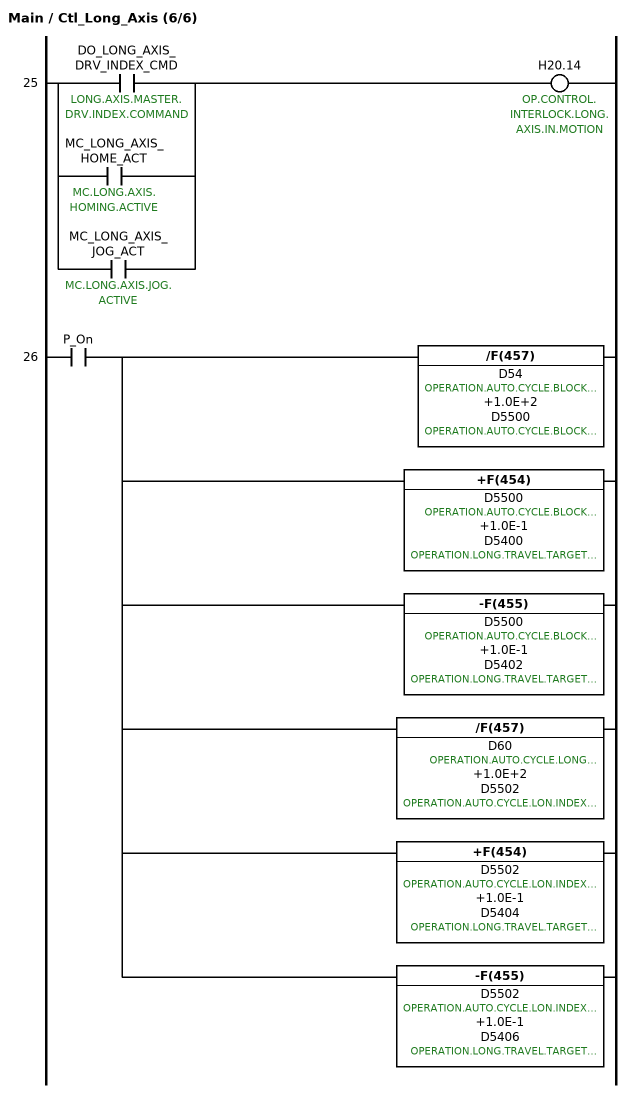
; rung 25
LD DO_LONG_AXIS_DRV_INDEX_CMD  ; LONG.AXIS.MASTER.DRV.INDEX.COMMAND
OR MC_LONG_AXIS_HOME_ACT  ; MC.LONG.AXIS.HOMING.ACTIVE
OR MC_LONG_AXIS_JOG_ACT  ; MC.LONG.AXIS.JOG.ACTIVE
OUT H20.14  ; OP.CONTROL.INTERLOCK.LONG.AXIS.IN.MOTION
; rung 26
LD P_On
/F(457) D54 +1.0E+2 D5500  ; OPERATION.AUTO.CYCLE.BLOCK.FIRST.CUT.REAL, OPERATION.AUTO.CYCLE.BLOCK.FIRST.CUT.REAL.SCALED
+F(454) D5500 +1.0E-1 D5400  ; OPERATION.AUTO.CYCLE.BLOCK.FIRST.CUT.REAL.SCALED, OPERATION.LONG.TRAVEL.TARGET.WINDOW.PLUS
-F(455) D5500 +1.0E-1 D5402  ; OPERATION.AUTO.CYCLE.BLOCK.FIRST.CUT.REAL.SCALED, OPERATION.LONG.TRAVEL.TARGET.WINDOW.MINUS
/F(457) D60 +1.0E+2 D5502  ; OPERATION.AUTO.CYCLE.LONG.INDEX.LOCATION.REAL, OPERATION.AUTO.CYCLE.LON.INDEX.LOCATION.REAL.SCALED
+F(454) D5502 +1.0E-1 D5404  ; OPERATION.AUTO.CYCLE.LON.INDEX.LOCATION.REAL.SCALED, OPERATION.LONG.TRAVEL.TARGET.WINDOW.SLABCUT.PLUS
-F(455) D5502 +1.0E-1 D5406  ; OPERATION.AUTO.CYCLE.LON.INDEX.LOCATION.REAL.SCALED, OPERATION.LONG.TRAVEL.TARGET.SLABCUT.MINUS

### Section Ctl_Vertical_Axis

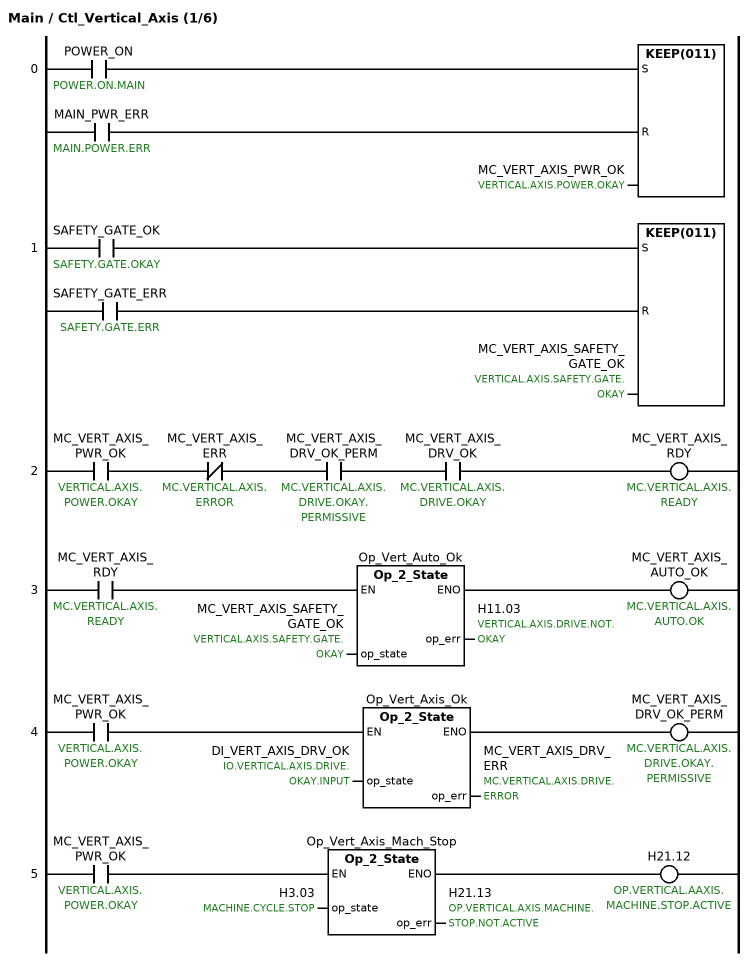
; rung 0
LD POWER_ON  ; POWER.ON.MAIN
LD MAIN_PWR_ERR  ; MAIN.POWER.ERR
KEEP(011) MC_VERT_AXIS_PWR_OK  ; VERTICAL.AXIS.POWER.OKAY
; rung 1
LD SAFETY_GATE_OK  ; SAFETY.GATE.OKAY
LD SAFETY_GATE_ERR  ; SAFETY.GATE.ERR
KEEP(011) MC_VERT_AXIS_SAFETY_GATE_OK  ; VERTICAL.AXIS.SAFETY.GATE.OKAY
; rung 2
LD MC_VERT_AXIS_PWR_OK  ; VERTICAL.AXIS.POWER.OKAY
ANDNOT MC_VERT_AXIS_ERR  ; MC.VERTICAL.AXIS.ERROR
AND MC_VERT_AXIS_DRV_OK_PERM  ; MC.VERTICAL.AXIS.DRIVE.OKAY.PERMISSIVE
AND MC_VERT_AXIS_DRV_OK  ; MC.VERTICAL.AXIS.DRIVE.OKAY
OUT MC_VERT_AXIS_RDY  ; MC.VERTICAL.AXIS.READY
; rung 3
LD MC_VERT_AXIS_RDY  ; MC.VERTICAL.AXIS.READY
CALL Op_Vert_Auto_Ok : Op_2_State (op_state := MC_VERT_AXIS_SAFETY_GATE_OK, op_err => H11.03)  ; VERTICAL.AXIS.SAFETY.GATE.OKAY, VERTICAL.AXIS.DRIVE.NOT.OKAY
OUT MC_VERT_AXIS_AUTO_OK  ; MC.VERTICAL.AXIS.AUTO.OK
; rung 4
LD MC_VERT_AXIS_PWR_OK  ; VERTICAL.AXIS.POWER.OKAY
CALL Op_Vert_Axis_Ok : Op_2_State (op_state := DI_VERT_AXIS_DRV_OK, op_err => MC_VERT_AXIS_DRV_ERR)  ; IO.VERTICAL.AXIS.DRIVE.OKAY.INPUT, MC.VERTICAL.AXIS.DRIVE.ERROR
OUT MC_VERT_AXIS_DRV_OK_PERM  ; MC.VERTICAL.AXIS.DRIVE.OKAY.PERMISSIVE
; rung 5
LD MC_VERT_AXIS_PWR_OK  ; VERTICAL.AXIS.POWER.OKAY
CALL Op_Vert_Axis_Mach_Stop : Op_2_State (op_state := H3.03, op_err => H21.13)  ; MACHINE.CYCLE.STOP, OP.VERTICAL.AXIS.MACHINE.STOP.NOT.ACTIVE
OUT H21.12  ; OP.VERTICAL.AAXIS.MACHINE.STOP.ACTIVE

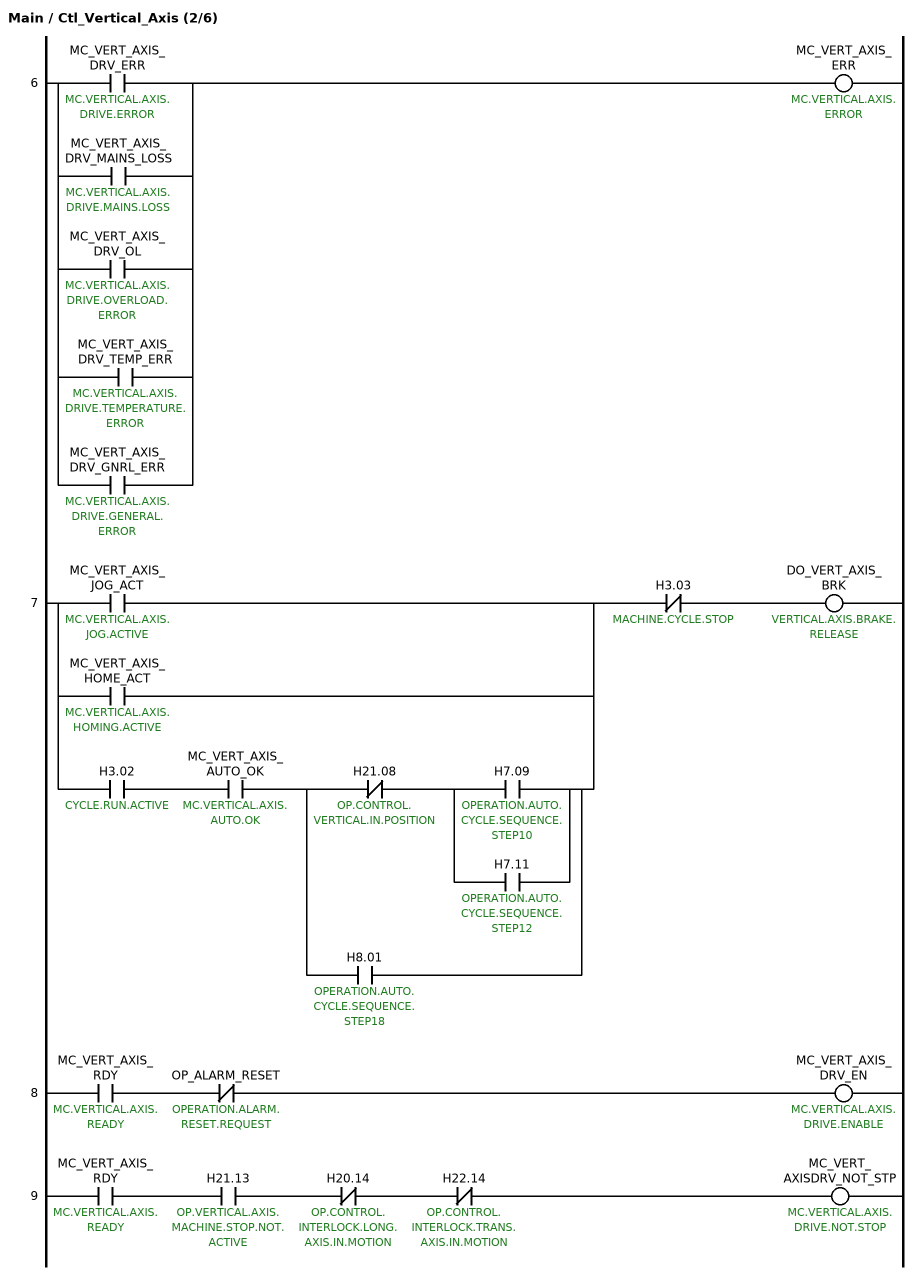
; rung 6
LD MC_VERT_AXIS_DRV_ERR  ; MC.VERTICAL.AXIS.DRIVE.ERROR
OR MC_VERT_AXIS_DRV_MAINS_LOSS  ; MC.VERTICAL.AXIS.DRIVE.MAINS.LOSS
OR MC_VERT_AXIS_DRV_OL  ; MC.VERTICAL.AXIS.DRIVE.OVERLOAD.ERROR
OR MC_VERT_AXIS_DRV_TEMP_ERR  ; MC.VERTICAL.AXIS.DRIVE.TEMPERATURE.ERROR
OR MC_VERT_AXIS_DRV_GNRL_ERR  ; MC.VERTICAL.AXIS.DRIVE.GENERAL.ERROR
OUT MC_VERT_AXIS_ERR  ; MC.VERTICAL.AXIS.ERROR
; rung 7
LD MC_VERT_AXIS_JOG_ACT  ; MC.VERTICAL.AXIS.JOG.ACTIVE
OR MC_VERT_AXIS_HOME_ACT  ; MC.VERTICAL.AXIS.HOMING.ACTIVE
LD H3.02  ; CYCLE.RUN.ACTIVE
AND MC_VERT_AXIS_AUTO_OK  ; MC.VERTICAL.AXIS.AUTO.OK
LDNOT H21.08  ; OP.CONTROL.VERTICAL.IN.POSITION
LD H7.09  ; OPERATION.AUTO.CYCLE.SEQUENCE.STEP10
OR H7.11  ; OPERATION.AUTO.CYCLE.SEQUENCE.STEP12
ANDLD
OR H8.01  ; OPERATION.AUTO.CYCLE.SEQUENCE.STEP18
ANDLD
ORLD
ANDNOT H3.03  ; MACHINE.CYCLE.STOP
OUT DO_VERT_AXIS_BRK  ; VERTICAL.AXIS.BRAKE.RELEASE
; rung 8
LD MC_VERT_AXIS_RDY  ; MC.VERTICAL.AXIS.READY
ANDNOT OP_ALARM_RESET  ; OPERATION.ALARM.RESET.REQUEST
OUT MC_VERT_AXIS_DRV_EN  ; MC.VERTICAL.AXIS.DRIVE.ENABLE
; rung 9
LD MC_VERT_AXIS_RDY  ; MC.VERTICAL.AXIS.READY
AND H21.13  ; OP.VERTICAL.AXIS.MACHINE.STOP.NOT.ACTIVE
ANDNOT H20.14  ; OP.CONTROL.INTERLOCK.LONG.AXIS.IN.MOTION
ANDNOT H22.14  ; OP.CONTROL.INTERLOCK.TRANS.AXIS.IN.MOTION
OUT MC_VERT_AXISDRV_NOT_STP  ; MC.VERTICAL.AXIS.DRIVE.NOT.STOP

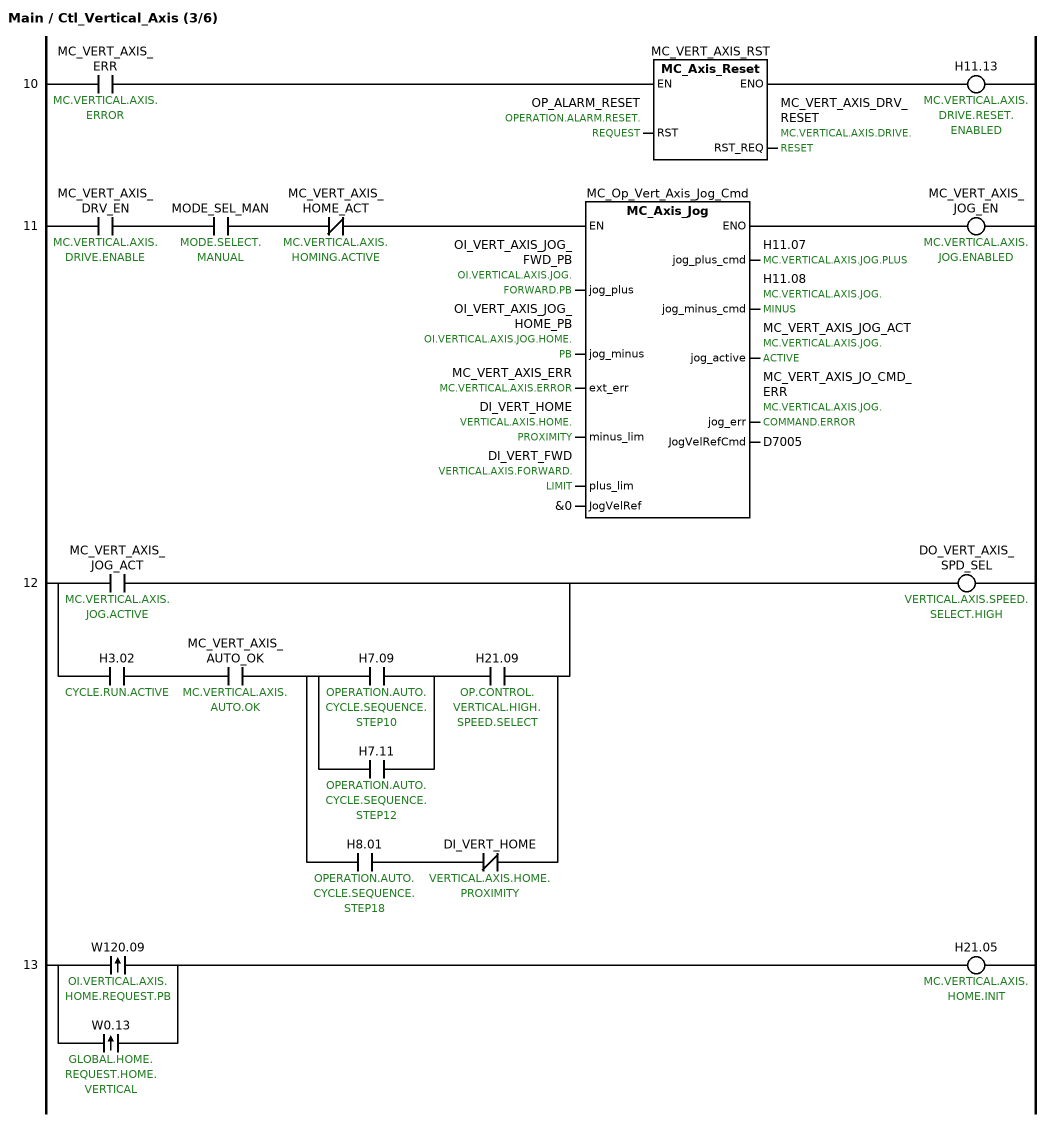
; rung 10
LD MC_VERT_AXIS_ERR  ; MC.VERTICAL.AXIS.ERROR
CALL MC_VERT_AXIS_RST : MC_Axis_Reset (RST := OP_ALARM_RESET, RST_REQ => MC_VERT_AXIS_DRV_RESET)  ; OPERATION.ALARM.RESET.REQUEST, MC.VERTICAL.AXIS.DRIVE.RESET
OUT H11.13  ; MC.VERTICAL.AXIS.DRIVE.RESET.ENABLED
; rung 11
LD MC_VERT_AXIS_DRV_EN  ; MC.VERTICAL.AXIS.DRIVE.ENABLE
AND MODE_SEL_MAN  ; MODE.SELECT.MANUAL
ANDNOT MC_VERT_AXIS_HOME_ACT  ; MC.VERTICAL.AXIS.HOMING.ACTIVE
CALL MC_Op_Vert_Axis_Jog_Cmd : MC_Axis_Jog (jog_plus := OI_VERT_AXIS_JOG_FWD_PB, jog_minus := OI_VERT_AXIS_JOG_HOME_PB, ext_err := MC_VERT_AXIS_ERR, minus_lim := DI_VERT_HOME, plus_lim := DI_VERT_FWD, JogVelRef := &0, jog_plus_cmd => H11.07, jog_minus_cmd => H11.08, jog_active => MC_VERT_AXIS_JOG_ACT, jog_err => MC_VERT_AXIS_JO_CMD_ERR, JogVelRefCmd => D7005)  ; OI.VERTICAL.AXIS.JOG.FORWARD.PB, OI.VERTICAL.AXIS.JOG.HOME.PB, MC.VERTICAL.AXIS.ERROR, VERTICAL.AXIS.HOME.PROXIMITY, VERTICAL.AXIS.FORWARD.LIMIT, MC.VERTICAL.AXIS.JOG.PLUS, MC.VERTICAL.AXIS.JOG.MINUS, MC.VERTICAL.AXIS.JOG.ACTIVE, MC.VERTICAL.AXIS.JOG.COMMAND.ERROR
OUT MC_VERT_AXIS_JOG_EN  ; MC.VERTICAL.AXIS.JOG.ENABLED
; rung 12
LD MC_VERT_AXIS_JOG_ACT  ; MC.VERTICAL.AXIS.JOG.ACTIVE
LD H3.02  ; CYCLE.RUN.ACTIVE
AND MC_VERT_AXIS_AUTO_OK  ; MC.VERTICAL.AXIS.AUTO.OK
LD H7.09  ; OPERATION.AUTO.CYCLE.SEQUENCE.STEP10
OR H7.11  ; OPERATION.AUTO.CYCLE.SEQUENCE.STEP12
AND H21.09  ; OP.CONTROL.VERTICAL.HIGH.SPEED.SELECT
LD H8.01  ; OPERATION.AUTO.CYCLE.SEQUENCE.STEP18
ANDNOT DI_VERT_HOME  ; VERTICAL.AXIS.HOME.PROXIMITY
ORLD
ANDLD
ORLD
OUT DO_VERT_AXIS_SPD_SEL  ; VERTICAL.AXIS.SPEED.SELECT.HIGH
; rung 13
@LD W120.09  ; OI.VERTICAL.AXIS.HOME.REQUEST.PB
@OR W0.13  ; GLOBAL.HOME.REQUEST.HOME.VERTICAL
OUT H21.05  ; MC.VERTICAL.AXIS.HOME.INIT

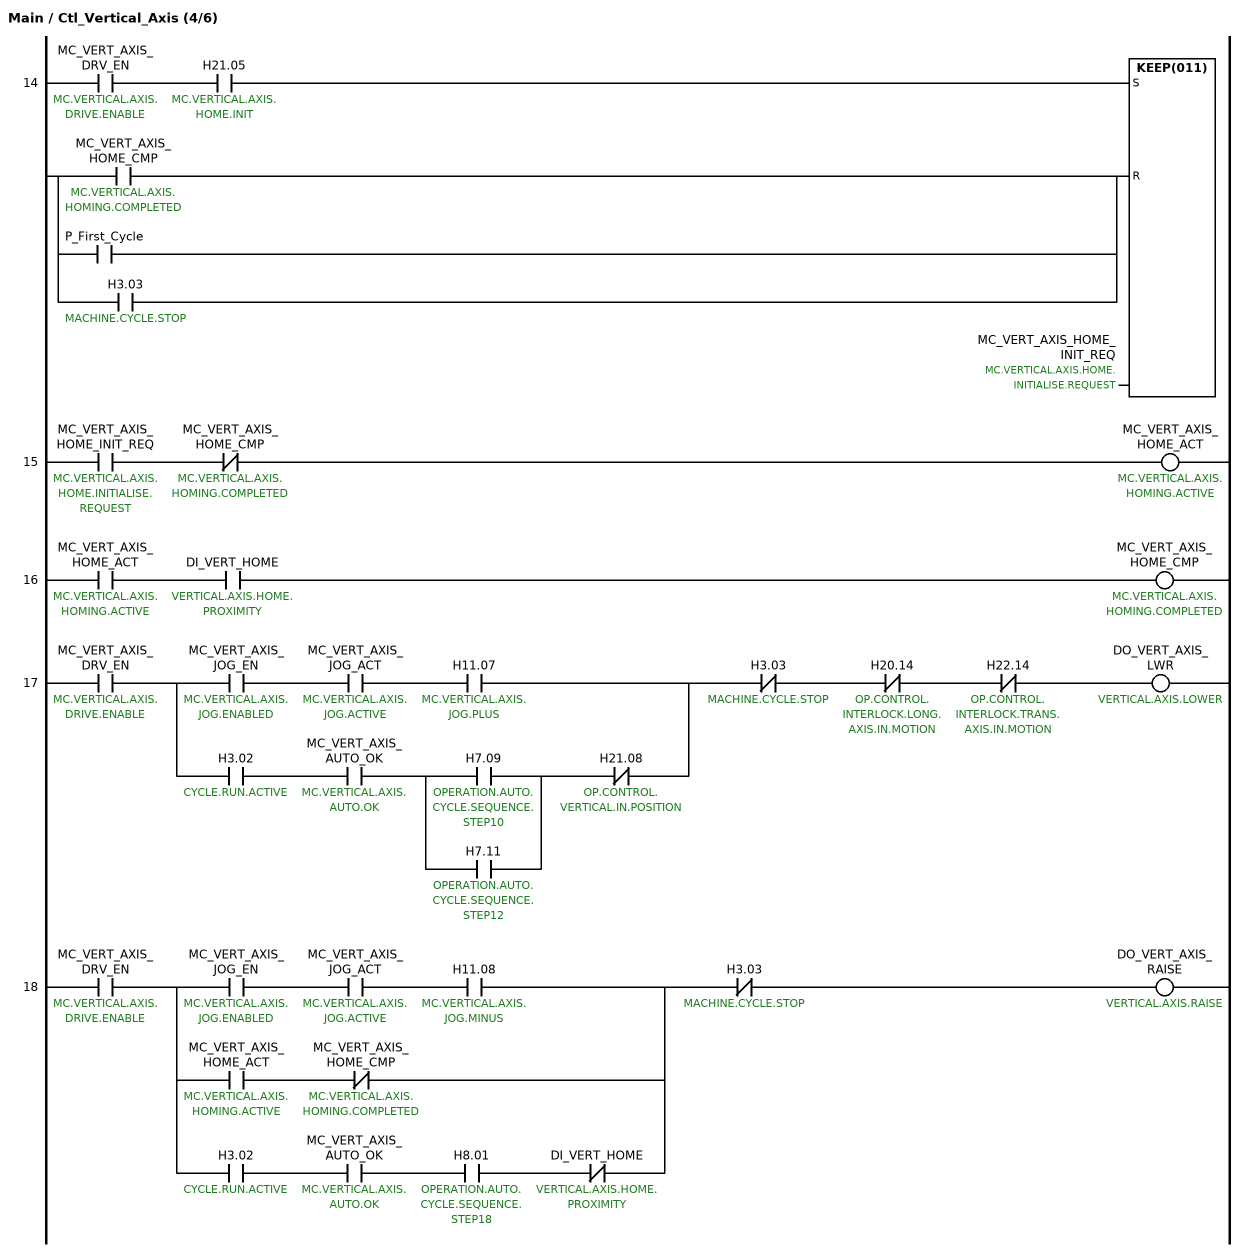
; rung 14
LD MC_VERT_AXIS_DRV_EN  ; MC.VERTICAL.AXIS.DRIVE.ENABLE
AND H21.05  ; MC.VERTICAL.AXIS.HOME.INIT
LD MC_VERT_AXIS_HOME_CMP  ; MC.VERTICAL.AXIS.HOMING.COMPLETED
OR P_First_Cycle
OR H3.03  ; MACHINE.CYCLE.STOP
KEEP(011) MC_VERT_AXIS_HOME_INIT_REQ  ; MC.VERTICAL.AXIS.HOME.INITIALISE.REQUEST
; rung 15
LD MC_VERT_AXIS_HOME_INIT_REQ  ; MC.VERTICAL.AXIS.HOME.INITIALISE.REQUEST
ANDNOT MC_VERT_AXIS_HOME_CMP  ; MC.VERTICAL.AXIS.HOMING.COMPLETED
OUT MC_VERT_AXIS_HOME_ACT  ; MC.VERTICAL.AXIS.HOMING.ACTIVE
; rung 16
LD MC_VERT_AXIS_HOME_ACT  ; MC.VERTICAL.AXIS.HOMING.ACTIVE
AND DI_VERT_HOME  ; VERTICAL.AXIS.HOME.PROXIMITY
OUT MC_VERT_AXIS_HOME_CMP  ; MC.VERTICAL.AXIS.HOMING.COMPLETED
; rung 17
LD MC_VERT_AXIS_DRV_EN  ; MC.VERTICAL.AXIS.DRIVE.ENABLE
LD MC_VERT_AXIS_JOG_EN  ; MC.VERTICAL.AXIS.JOG.ENABLED
AND MC_VERT_AXIS_JOG_ACT  ; MC.VERTICAL.AXIS.JOG.ACTIVE
AND H11.07  ; MC.VERTICAL.AXIS.JOG.PLUS
LD H3.02  ; CYCLE.RUN.ACTIVE
AND MC_VERT_AXIS_AUTO_OK  ; MC.VERTICAL.AXIS.AUTO.OK
LD H7.09  ; OPERATION.AUTO.CYCLE.SEQUENCE.STEP10
OR H7.11  ; OPERATION.AUTO.CYCLE.SEQUENCE.STEP12
ANDLD
ANDNOT H21.08  ; OP.CONTROL.VERTICAL.IN.POSITION
ORLD
ANDLD
ANDNOT H3.03  ; MACHINE.CYCLE.STOP
ANDNOT H20.14  ; OP.CONTROL.INTERLOCK.LONG.AXIS.IN.MOTION
ANDNOT H22.14  ; OP.CONTROL.INTERLOCK.TRANS.AXIS.IN.MOTION
OUT DO_VERT_AXIS_LWR  ; VERTICAL.AXIS.LOWER
; rung 18
LD MC_VERT_AXIS_DRV_EN  ; MC.VERTICAL.AXIS.DRIVE.ENABLE
LD MC_VERT_AXIS_JOG_EN  ; MC.VERTICAL.AXIS.JOG.ENABLED
AND MC_VERT_AXIS_JOG_ACT  ; MC.VERTICAL.AXIS.JOG.ACTIVE
AND H11.08  ; MC.VERTICAL.AXIS.JOG.MINUS
LD MC_VERT_AXIS_HOME_ACT  ; MC.VERTICAL.AXIS.HOMING.ACTIVE
ANDNOT MC_VERT_AXIS_HOME_CMP  ; MC.VERTICAL.AXIS.HOMING.COMPLETED
ORLD
LD H3.02  ; CYCLE.RUN.ACTIVE
AND MC_VERT_AXIS_AUTO_OK  ; MC.VERTICAL.AXIS.AUTO.OK
AND H8.01  ; OPERATION.AUTO.CYCLE.SEQUENCE.STEP18
ANDNOT DI_VERT_HOME  ; VERTICAL.AXIS.HOME.PROXIMITY
ORLD
ANDLD
ANDNOT H3.03  ; MACHINE.CYCLE.STOP
OUT DO_VERT_AXIS_RAISE  ; VERTICAL.AXIS.RAISE

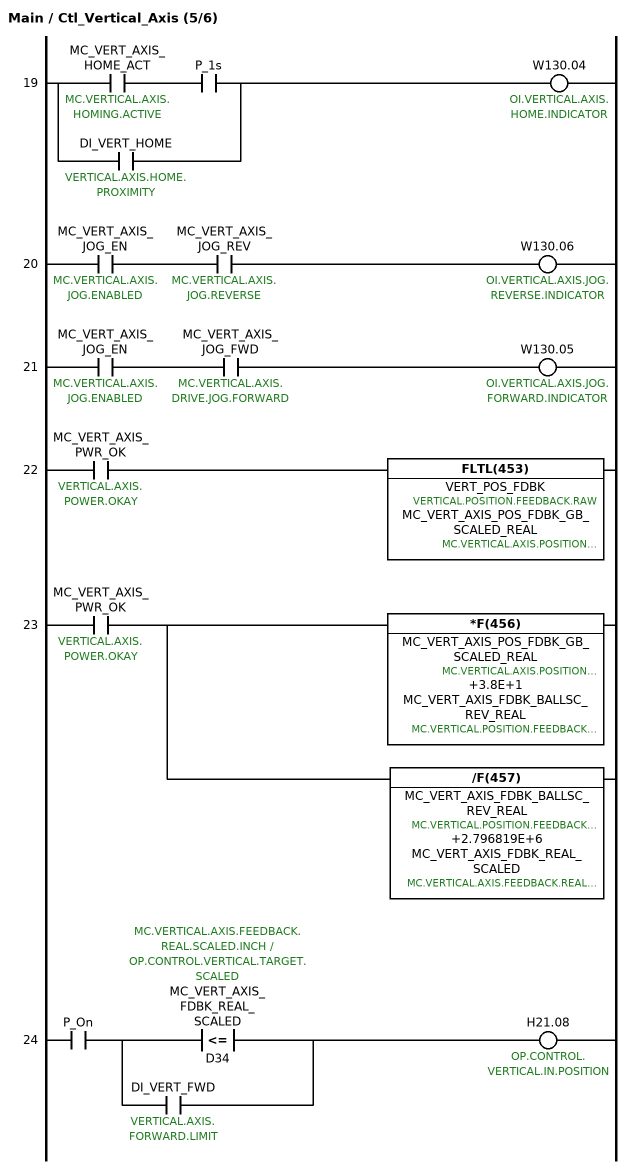
; rung 19
LD MC_VERT_AXIS_HOME_ACT  ; MC.VERTICAL.AXIS.HOMING.ACTIVE
AND P_1s
OR DI_VERT_HOME  ; VERTICAL.AXIS.HOME.PROXIMITY
OUT W130.04  ; OI.VERTICAL.AXIS.HOME.INDICATOR
; rung 20
LD MC_VERT_AXIS_JOG_EN  ; MC.VERTICAL.AXIS.JOG.ENABLED
AND MC_VERT_AXIS_JOG_REV  ; MC.VERTICAL.AXIS.JOG.REVERSE
OUT W130.06  ; OI.VERTICAL.AXIS.JOG.REVERSE.INDICATOR
; rung 21
LD MC_VERT_AXIS_JOG_EN  ; MC.VERTICAL.AXIS.JOG.ENABLED
AND MC_VERT_AXIS_JOG_FWD  ; MC.VERTICAL.AXIS.DRIVE.JOG.FORWARD
OUT W130.05  ; OI.VERTICAL.AXIS.JOG.FORWARD.INDICATOR
; rung 22
LD MC_VERT_AXIS_PWR_OK  ; VERTICAL.AXIS.POWER.OKAY
FLTL(453) VERT_POS_FDBK MC_VERT_AXIS_POS_FDBK_GB_SCALED_REAL  ; VERTICAL.POSITION.FEEDBACK.RAW, MC.VERTICAL.AXIS.POSITION.REVOLUTION.REAL
; rung 23
LD MC_VERT_AXIS_PWR_OK  ; VERTICAL.AXIS.POWER.OKAY
*F(456) MC_VERT_AXIS_POS_FDBK_GB_SCALED_REAL +3.8E+1 MC_VERT_AXIS_FDBK_BALLSC_REV_REAL  ; MC.VERTICAL.AXIS.POSITION.REVOLUTION.REAL, MC.VERTICAL.POSITION.FEEDBACK.BALLSCREW.REVOLUTIONS.REAL
/F(457) MC_VERT_AXIS_FDBK_BALLSC_REV_REAL +2.796819E+6 MC_VERT_AXIS_FDBK_REAL_SCALED  ; MC.VERTICAL.POSITION.FEEDBACK.BALLSCREW.REVOLUTIONS.REAL, MC.VERTICAL.AXIS.FEEDBACK.REAL.SCALED.INCH
; rung 24
LD P_On
LD<=F(332) MC_VERT_AXIS_FDBK_REAL_SCALED D34  ; MC.VERTICAL.AXIS.FEEDBACK.REAL.SCALED.INCH, OP.CONTROL.VERTICAL.TARGET.SCALED
OR DI_VERT_FWD  ; VERTICAL.AXIS.FORWARD.LIMIT
ANDLD
OUT H21.08  ; OP.CONTROL.VERTICAL.IN.POSITION

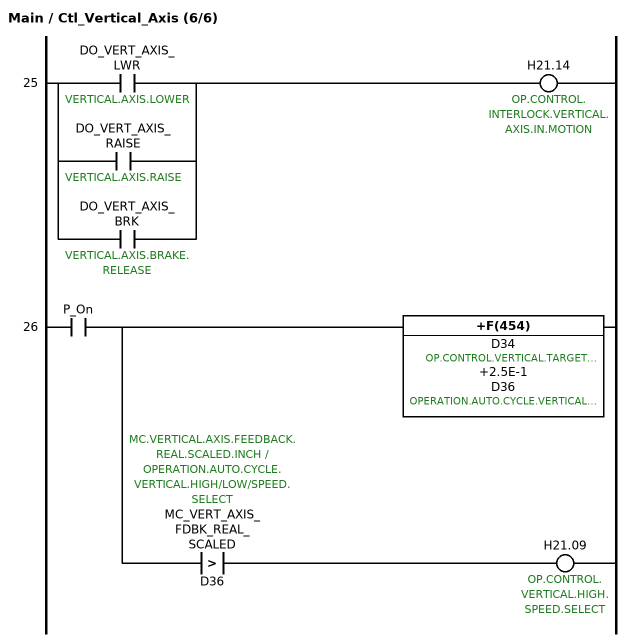
; rung 25
LD DO_VERT_AXIS_LWR  ; VERTICAL.AXIS.LOWER
OR DO_VERT_AXIS_RAISE  ; VERTICAL.AXIS.RAISE
OR DO_VERT_AXIS_BRK  ; VERTICAL.AXIS.BRAKE.RELEASE
OUT H21.14  ; OP.CONTROL.INTERLOCK.VERTICAL.AXIS.IN.MOTION
; rung 26
LD P_On
+F(454) D34 +2.5E-1 D36  ; OP.CONTROL.VERTICAL.TARGET.SCALED, OPERATION.AUTO.CYCLE.VERTICAL.HIGH/LOW/SPEED.SELECT
AND>F(333) MC_VERT_AXIS_FDBK_REAL_SCALED D36  ; MC.VERTICAL.AXIS.FEEDBACK.REAL.SCALED.INCH, OPERATION.AUTO.CYCLE.VERTICAL.HIGH/LOW/SPEED.SELECT
OUT H21.09  ; OP.CONTROL.VERTICAL.HIGH.SPEED.SELECT

### Section Ctl_Transverse_Axis

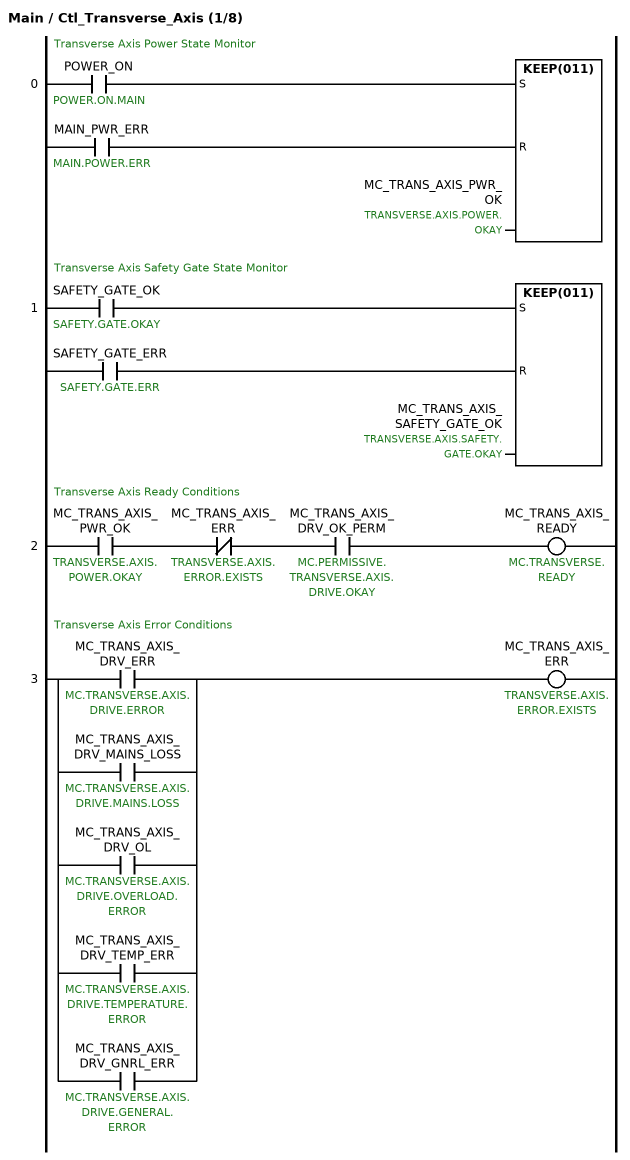
; rung 0: Transverse Axis Power State Monitor
LD POWER_ON  ; POWER.ON.MAIN
LD MAIN_PWR_ERR  ; MAIN.POWER.ERR
KEEP(011) MC_TRANS_AXIS_PWR_OK  ; TRANSVERSE.AXIS.POWER.OKAY
; rung 1: Transverse Axis Safety Gate State Monitor
LD SAFETY_GATE_OK  ; SAFETY.GATE.OKAY
LD SAFETY_GATE_ERR  ; SAFETY.GATE.ERR
KEEP(011) MC_TRANS_AXIS_SAFETY_GATE_OK  ; TRANSVERSE.AXIS.SAFETY.GATE.OKAY
; rung 2: Transverse Axis Ready Conditions
LD MC_TRANS_AXIS_PWR_OK  ; TRANSVERSE.AXIS.POWER.OKAY
ANDNOT MC_TRANS_AXIS_ERR  ; TRANSVERSE.AXIS.ERROR.EXISTS
AND MC_TRANS_AXIS_DRV_OK_PERM  ; MC.PERMISSIVE.TRANSVERSE.AXIS.DRIVE.OKAY
OUT MC_TRANS_AXIS_READY  ; MC.TRANSVERSE.READY
; rung 3: Transverse Axis Error Conditions
LD MC_TRANS_AXIS_DRV_ERR  ; MC.TRANSVERSE.AXIS.DRIVE.ERROR
OR MC_TRANS_AXIS_DRV_MAINS_LOSS  ; MC.TRANSVERSE.AXIS.DRIVE.MAINS.LOSS
OR MC_TRANS_AXIS_DRV_OL  ; MC.TRANSVERSE.AXIS.DRIVE.OVERLOAD.ERROR
OR MC_TRANS_AXIS_DRV_TEMP_ERR  ; MC.TRANSVERSE.AXIS.DRIVE.TEMPERATURE.ERROR
OR MC_TRANS_AXIS_DRV_GNRL_ERR  ; MC.TRANSVERSE.AXIS.DRIVE.GENERAL.ERROR
OUT MC_TRANS_AXIS_ERR  ; TRANSVERSE.AXIS.ERROR.EXISTS

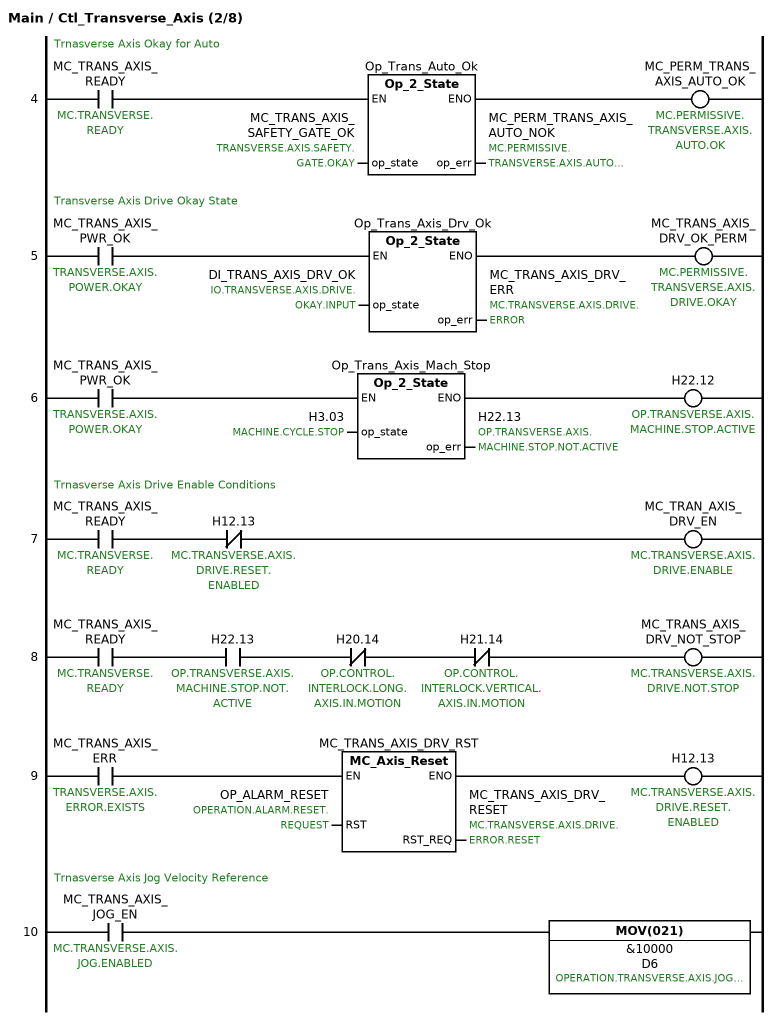
; rung 4: Trnasverse Axis Okay for Auto
LD MC_TRANS_AXIS_READY  ; MC.TRANSVERSE.READY
CALL Op_Trans_Auto_Ok : Op_2_State (op_state := MC_TRANS_AXIS_SAFETY_GATE_OK, op_err => MC_PERM_TRANS_AXIS_AUTO_NOK)  ; TRANSVERSE.AXIS.SAFETY.GATE.OKAY, MC.PERMISSIVE.TRANSVERSE.AXIS.AUTO.NOK
OUT MC_PERM_TRANS_AXIS_AUTO_OK  ; MC.PERMISSIVE.TRANSVERSE.AXIS.AUTO.OK
; rung 5: Transverse Axis Drive Okay State
LD MC_TRANS_AXIS_PWR_OK  ; TRANSVERSE.AXIS.POWER.OKAY
CALL Op_Trans_Axis_Drv_Ok : Op_2_State (op_state := DI_TRANS_AXIS_DRV_OK, op_err => MC_TRANS_AXIS_DRV_ERR)  ; IO.TRANSVERSE.AXIS.DRIVE.OKAY.INPUT, MC.TRANSVERSE.AXIS.DRIVE.ERROR
OUT MC_TRANS_AXIS_DRV_OK_PERM  ; MC.PERMISSIVE.TRANSVERSE.AXIS.DRIVE.OKAY
; rung 6
LD MC_TRANS_AXIS_PWR_OK  ; TRANSVERSE.AXIS.POWER.OKAY
CALL Op_Trans_Axis_Mach_Stop : Op_2_State (op_state := H3.03, op_err => H22.13)  ; MACHINE.CYCLE.STOP, OP.TRANSVERSE.AXIS.MACHINE.STOP.NOT.ACTIVE
OUT H22.12  ; OP.TRANSVERSE.AXIS.MACHINE.STOP.ACTIVE
; rung 7: Trnasverse Axis Drive Enable Conditions
LD MC_TRANS_AXIS_READY  ; MC.TRANSVERSE.READY
ANDNOT H12.13  ; MC.TRANSVERSE.AXIS.DRIVE.RESET.ENABLED
OUT MC_TRAN_AXIS_DRV_EN  ; MC.TRANSVERSE.AXIS.DRIVE.ENABLE
; rung 8
LD MC_TRANS_AXIS_READY  ; MC.TRANSVERSE.READY
AND H22.13  ; OP.TRANSVERSE.AXIS.MACHINE.STOP.NOT.ACTIVE
ANDNOT H20.14  ; OP.CONTROL.INTERLOCK.LONG.AXIS.IN.MOTION
ANDNOT H21.14  ; OP.CONTROL.INTERLOCK.VERTICAL.AXIS.IN.MOTION
OUT MC_TRANS_AXIS_DRV_NOT_STOP  ; MC.TRANSVERSE.AXIS.DRIVE.NOT.STOP
; rung 9
LD MC_TRANS_AXIS_ERR  ; TRANSVERSE.AXIS.ERROR.EXISTS
CALL MC_TRANS_AXIS_DRV_RST : MC_Axis_Reset (RST := OP_ALARM_RESET, RST_REQ => MC_TRANS_AXIS_DRV_RESET)  ; OPERATION.ALARM.RESET.REQUEST, MC.TRANSVERSE.AXIS.DRIVE.ERROR.RESET
OUT H12.13  ; MC.TRANSVERSE.AXIS.DRIVE.RESET.ENABLED
; rung 10: Trnasverse Axis Jog Velocity Reference
LD MC_TRANS_AXIS_JOG_EN  ; MC.TRANSVERSE.AXIS.JOG.ENABLED
MOV(021) &10000 D6  ; OPERATION.TRANSVERSE.AXIS.JOG.VELOCITY.REFERNCE.WORD

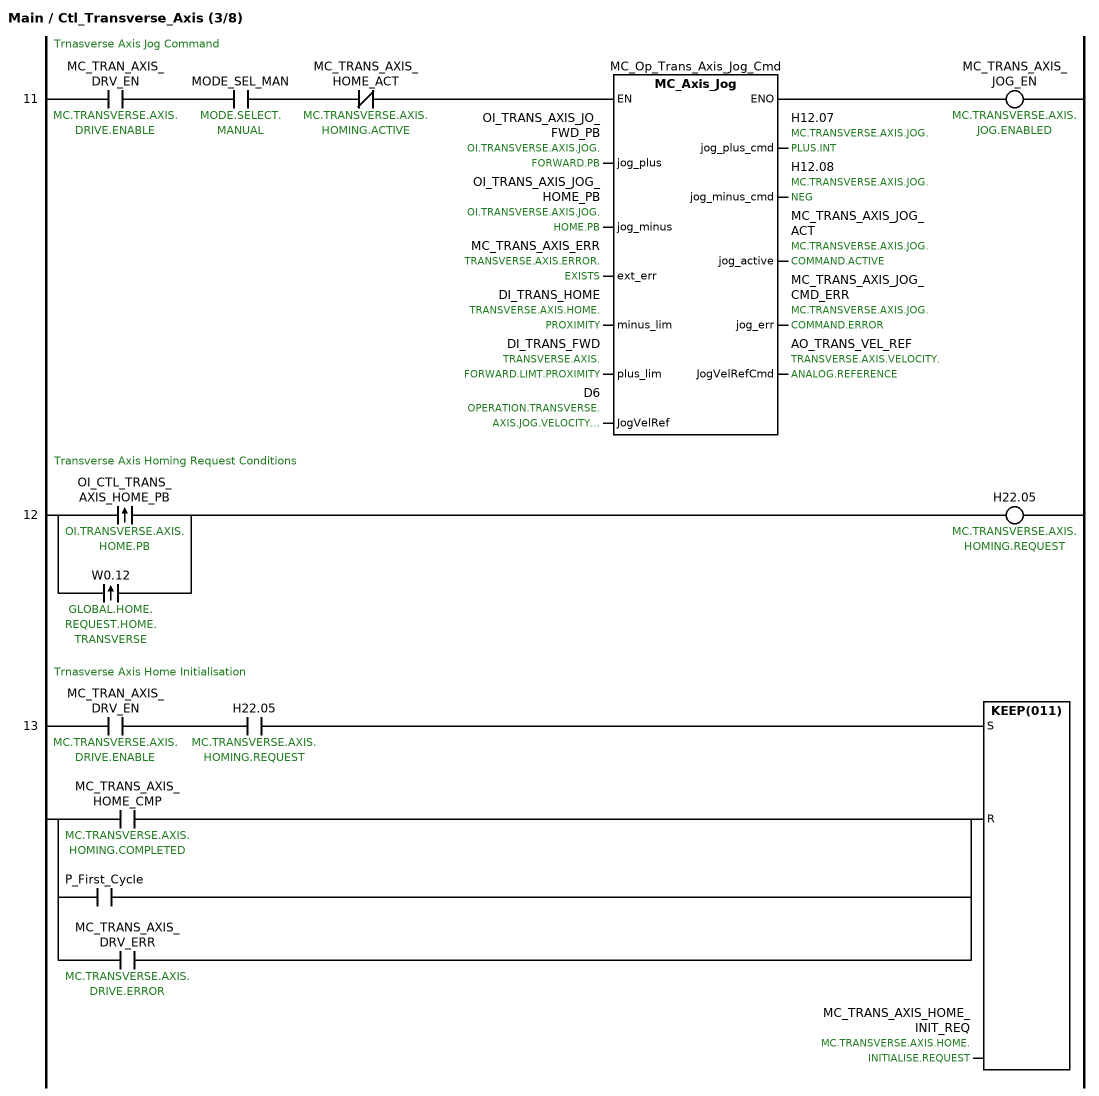
; rung 11: Trnasverse Axis Jog Command
LD MC_TRAN_AXIS_DRV_EN  ; MC.TRANSVERSE.AXIS.DRIVE.ENABLE
AND MODE_SEL_MAN  ; MODE.SELECT.MANUAL
ANDNOT MC_TRANS_AXIS_HOME_ACT  ; MC.TRANSVERSE.AXIS.HOMING.ACTIVE
CALL MC_Op_Trans_Axis_Jog_Cmd : MC_Axis_Jog (jog_plus := OI_TRANS_AXIS_JO_FWD_PB, jog_minus := OI_TRANS_AXIS_JOG_HOME_PB, ext_err := MC_TRANS_AXIS_ERR, minus_lim := DI_TRANS_HOME, plus_lim := DI_TRANS_FWD, JogVelRef := D6, jog_plus_cmd => H12.07, jog_minus_cmd => H12.08, jog_active => MC_TRANS_AXIS_JOG_ACT, jog_err => MC_TRANS_AXIS_JOG_CMD_ERR, JogVelRefCmd => AO_TRANS_VEL_REF)  ; OI.TRANSVERSE.AXIS.JOG.FORWARD.PB, OI.TRANSVERSE.AXIS.JOG.HOME.PB, TRANSVERSE.AXIS.ERROR.EXISTS, TRANSVERSE.AXIS.HOME.PROXIMITY, TRANSVERSE.AXIS.FORWARD.LIMT.PROXIMITY, OPERATION.TRANSVERSE.AXIS.JOG.VELOCITY.REFERNCE.WORD, MC.TRANSVERSE.AXIS.JOG.PLUS.INT, MC.TRANSVERSE.AXIS.JOG.NEG, MC.TRANSVERSE.AXIS.JOG.COMMAND.ACTIVE, MC.TRANSVERSE.AXIS.JOG.COMMAND.ERROR, TRANSVERSE.AXIS.VELOCITY.ANALOG.REFERENCE
OUT MC_TRANS_AXIS_JOG_EN  ; MC.TRANSVERSE.AXIS.JOG.ENABLED
; rung 12: Transverse Axis Homing Request Conditions
@LD OI_CTL_TRANS_AXIS_HOME_PB  ; OI.TRANSVERSE.AXIS.HOME.PB
@OR W0.12  ; GLOBAL.HOME.REQUEST.HOME.TRANSVERSE
OUT H22.05  ; MC.TRANSVERSE.AXIS.HOMING.REQUEST
; rung 13: Trnasverse Axis Home Initialisation
LD MC_TRAN_AXIS_DRV_EN  ; MC.TRANSVERSE.AXIS.DRIVE.ENABLE
AND H22.05  ; MC.TRANSVERSE.AXIS.HOMING.REQUEST
LD MC_TRANS_AXIS_HOME_CMP  ; MC.TRANSVERSE.AXIS.HOMING.COMPLETED
OR P_First_Cycle
OR MC_TRANS_AXIS_DRV_ERR  ; MC.TRANSVERSE.AXIS.DRIVE.ERROR
KEEP(011) MC_TRANS_AXIS_HOME_INIT_REQ  ; MC.TRANSVERSE.AXIS.HOME.INITIALISE.REQUEST

